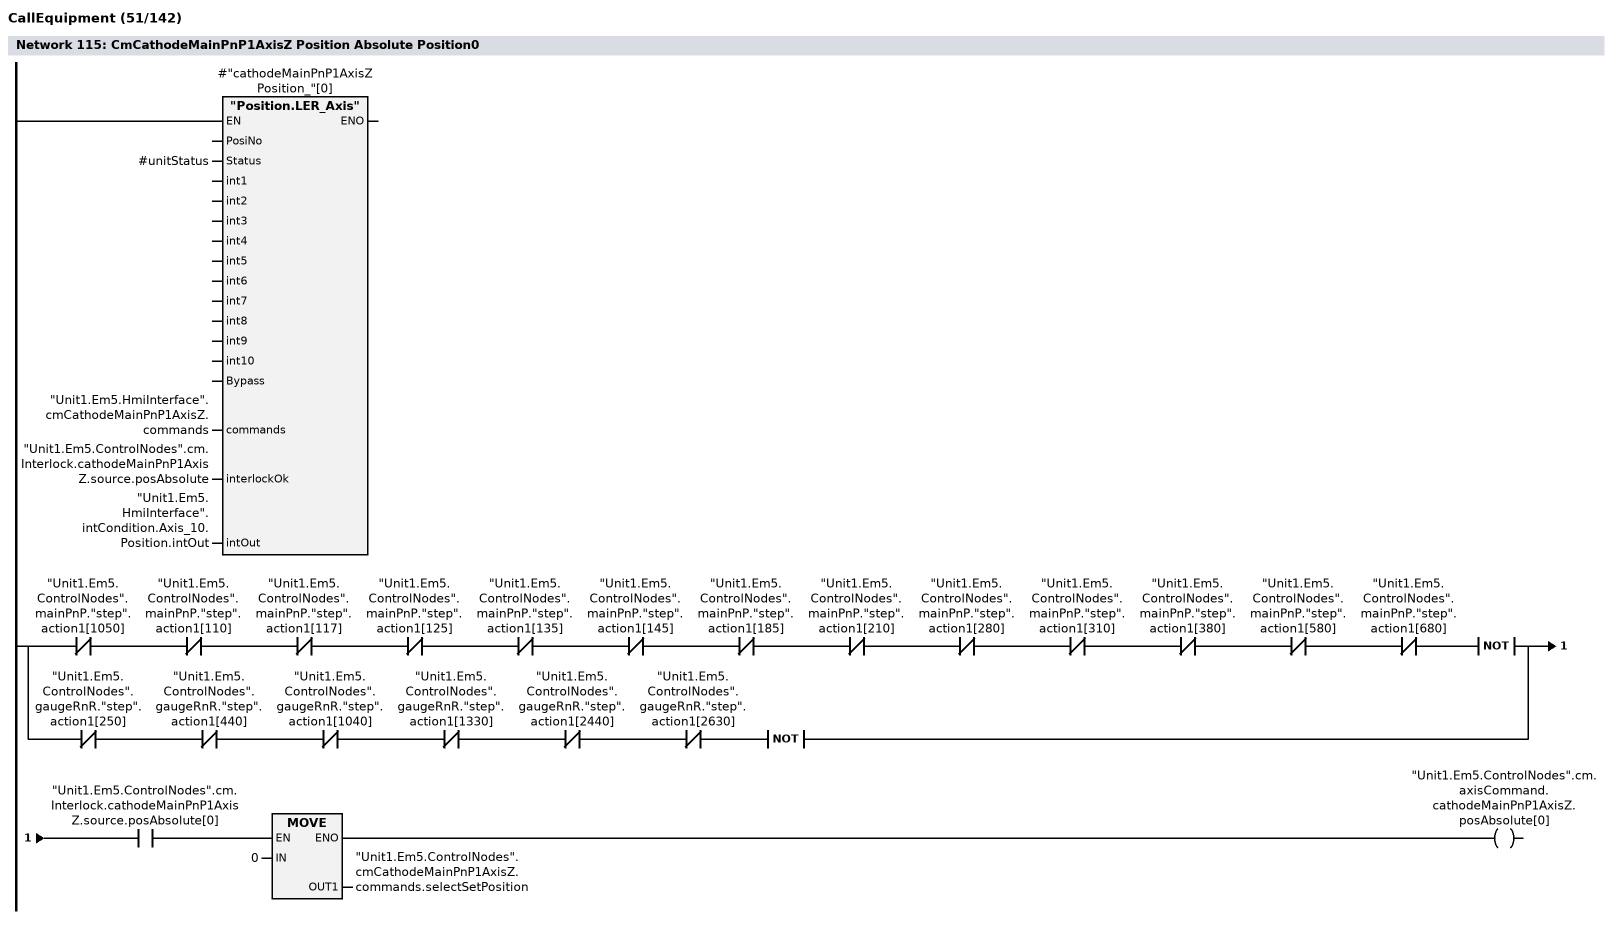
   RUNG wire#powerrail
      #"cathodeMainPnP1AxisZ Position_"[0](PosiNo :=, Status := #unitStatus, int1 :=, int2 :=, int3 :=, int4 :=, int5 :=, int6 :=, int7 :=, int8 :=, int9 :=, int10 :=, Bypass :=, commands := "Unit1.Em5.HmiInterface".cmCathodeMainPnP1AxisZ.commands, interlockOk := "Unit1.Em5.ControlNodes".cm.Interlock.cathodeMainPnP1AxisZ.source.posAbsolute, intOut := "Unit1.Em5.HmiInterface".intCondition.Axis_10.Position.intOut)
   END_RUNG
   RUNG wire#powerrail
      I_Contact( "Unit1.Em5.ControlNodes".mainPnP."step".action1[1050] )
      I_Contact( "Unit1.Em5.ControlNodes".mainPnP."step".action1[110] )
      I_Contact( "Unit1.Em5.ControlNodes".mainPnP."step".action1[117] )
      I_Contact( "Unit1.Em5.ControlNodes".mainPnP."step".action1[125] )
      I_Contact( "Unit1.Em5.ControlNodes".mainPnP."step".action1[135] )
      I_Contact( "Unit1.Em5.ControlNodes".mainPnP."step".action1[145] )
      I_Contact( "Unit1.Em5.ControlNodes".mainPnP."step".action1[185] )
      I_Contact( "Unit1.Em5.ControlNodes".mainPnP."step".action1[210] )
      I_Contact( "Unit1.Em5.ControlNodes".mainPnP."step".action1[280] )
      I_Contact( "Unit1.Em5.ControlNodes".mainPnP."step".action1[310] )
      I_Contact( "Unit1.Em5.ControlNodes".mainPnP."step".action1[380] )
      I_Contact( "Unit1.Em5.ControlNodes".mainPnP."step".action1[580] )
      I_Contact( "Unit1.Em5.ControlNodes".mainPnP."step".action1[680] )
      Not()
      wire#w1
      Contact( "Unit1.Em5.ControlNodes".cm.Interlock.cathodeMainPnP1AxisZ.source.posAbsolute[0] )
      Move(in := 0, out1 => "Unit1.Em5.ControlNodes".cmCathodeMainPnP1AxisZ.commands.selectSetPosition)
      Coil( "Unit1.Em5.ControlNodes".cm.axisCommand.cathodeMainPnP1AxisZ.posAbsolute[0] )
   END_RUNG
   RUNG wire#powerrail
      I_Contact( "Unit1.Em5.ControlNodes".gaugeRnR."step".action1[250] )
      I_Contact( "Unit1.Em5.ControlNodes".gaugeRnR."step".action1[440] )
      I_Contact( "Unit1.Em5.ControlNodes".gaugeRnR."step".action1[1040] )
      I_Contact( "Unit1.Em5.ControlNodes".gaugeRnR."step".action1[1330] )
      I_Contact( "Unit1.Em5.ControlNodes".gaugeRnR."step".action1[2440] )
      I_Contact( "Unit1.Em5.ControlNodes".gaugeRnR."step".action1[2630] )
      Not()
   END_RUNG wire#w1
   // the same network as SCL:
   #"cathodeMainPnP1AxisZ Position_"[0](Status := #unitStatus,   // "Position.LER_Axis"
                           commands := "Unit1.Em5.HmiInterface".cmCathodeMainPnP1AxisZ.commands,
                           interlockOk := "Unit1.Em5.ControlNodes".cm.Interlock.cathodeMainPnP1AxisZ.source.posAbsolute,
                           intOut := "Unit1.Em5.HmiInterface".intCondition.Axis_10.Position.intOut);
   #_w1 := (NOT (NOT "Unit1.Em5.ControlNodes".mainPnP."step".action1[1050] AND NOT "Unit1.Em5.ControlNodes".mainPnP."step".action1[110] AND NOT "Unit1.Em5.ControlNodes".mainPnP."step".action1[117] AND NOT "Unit1.Em5.ControlNodes".mainPnP."step".action1[125] AND NOT "Unit1.Em5.ControlNodes".mainPnP."step".action1[135] AND NOT "Unit1.Em5.ControlNodes".mainPnP."step".action1[145] AND NOT "Unit1.Em5.ControlNodes".mainPnP."step".action1[185] AND NOT "Unit1.Em5.ControlNodes".mainPnP."step".action1[210] AND NOT "Unit1.Em5.ControlNodes".mainPnP."step".action1[280] AND NOT "Unit1.Em5.ControlNodes".mainPnP."step".action1[310] AND NOT "Unit1.Em5.ControlNodes".mainPnP."step".action1[380] AND NOT "Unit1.Em5.ControlNodes".mainPnP."step".action1[580] AND NOT "Unit1.Em5.ControlNodes".mainPnP."step".action1[680]) OR NOT (NOT "Unit1.Em5.ControlNodes".gaugeRnR."step".action1[250] AND NOT "Unit1.Em5.ControlNodes".gaugeRnR."step".action1[440] AND NOT "Unit1.Em5.ControlNodes".gaugeRnR."step".action1[1040] AND NOT "Unit1.Em5.ControlNodes".gaugeRnR."step".action1[1330] AND NOT "Unit1.Em5.ControlNodes".gaugeRnR."step".action1[2440] AND NOT "Unit1.Em5.ControlNodes".gaugeRnR."step".action1[2630])) AND "Unit1.Em5.ControlNodes".cm.Interlock.cathodeMainPnP1AxisZ.source.posAbsolute[0];
   IF #_w1 THEN "Unit1.Em5.ControlNodes".cmCathodeMainPnP1AxisZ.commands.selectSetPosition := 0; END_IF;
   "Unit1.Em5.ControlNodes".cm.axisCommand.cathodeMainPnP1AxisZ.posAbsolute[0] := #_w1;
END_REGION

REGION Network 116: CmCathodeMainPnP1AxisZ Position Absolute Position1
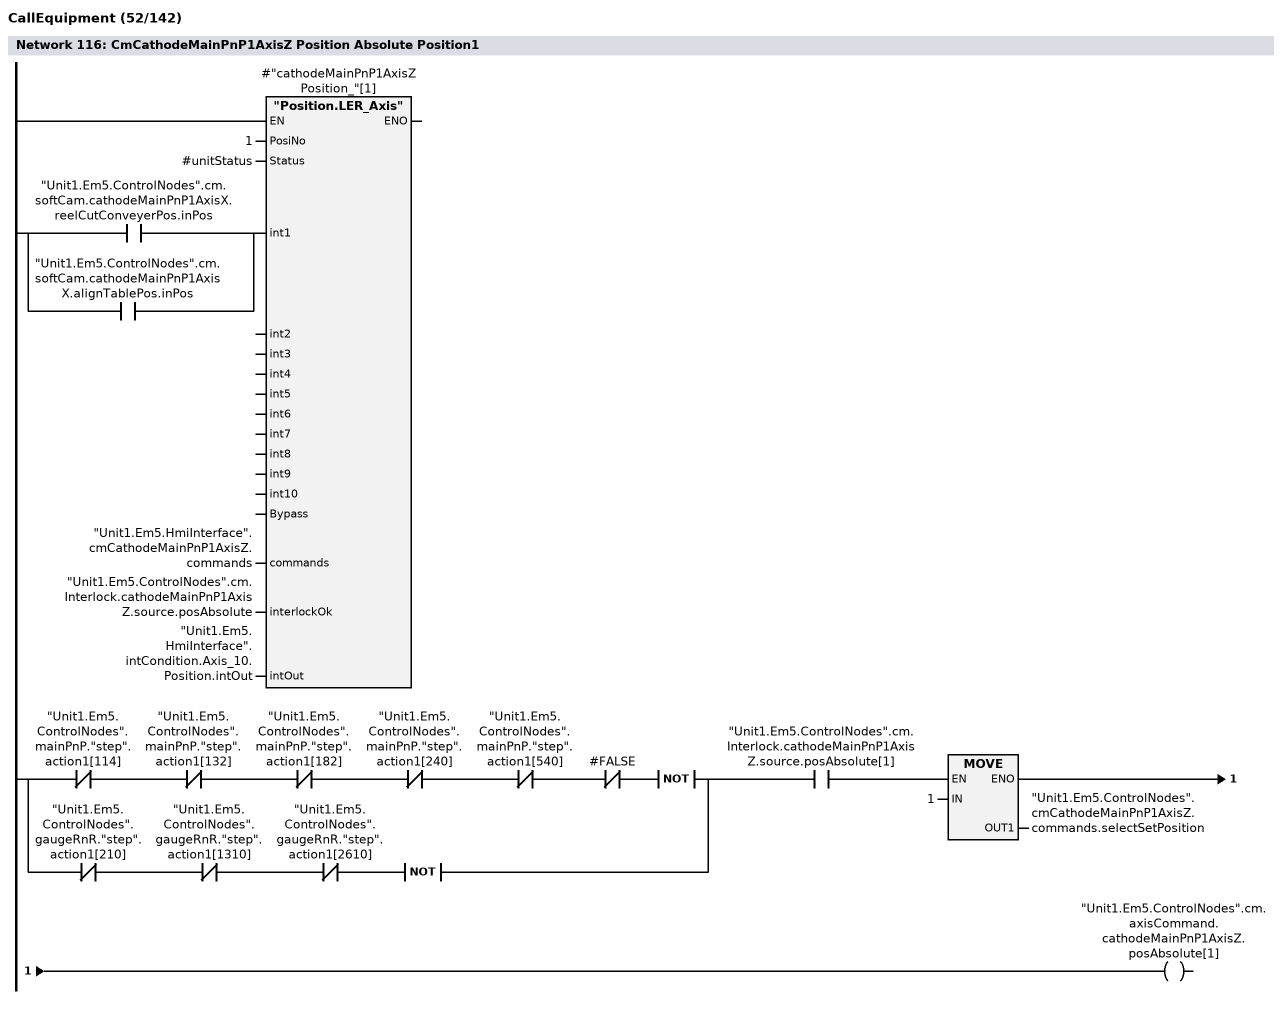
   RUNG wire#powerrail
      #"cathodeMainPnP1AxisZ Position_"[1](int1 := wire#w1, PosiNo := 1, Status := #unitStatus, int2 :=, int3 :=, int4 :=, int5 :=, int6 :=, int7 :=, int8 :=, int9 :=, int10 :=, Bypass :=, commands := "Unit1.Em5.HmiInterface".cmCathodeMainPnP1AxisZ.commands, interlockOk := "Unit1.Em5.ControlNodes".cm.Interlock.cathodeMainPnP1AxisZ.source.posAbsolute, intOut := "Unit1.Em5.HmiInterface".intCondition.Axis_10.Position.intOut)
   END_RUNG
   RUNG wire#powerrail
      Contact( "Unit1.Em5.ControlNodes".cm.softCam.cathodeMainPnP1AxisX.reelCutConveyerPos.inPos )
   END_RUNG wire#w1
   RUNG wire#powerrail
      Contact( "Unit1.Em5.ControlNodes".cm.softCam.cathodeMainPnP1AxisX.alignTablePos.inPos )
   END_RUNG wire#w1
   RUNG wire#powerrail
      I_Contact( "Unit1.Em5.ControlNodes".mainPnP."step".action1[114] )
      I_Contact( "Unit1.Em5.ControlNodes".mainPnP."step".action1[132] )
      I_Contact( "Unit1.Em5.ControlNodes".mainPnP."step".action1[182] )
      I_Contact( "Unit1.Em5.ControlNodes".mainPnP."step".action1[240] )
      I_Contact( "Unit1.Em5.ControlNodes".mainPnP."step".action1[540] )
      I_Contact( #FALSE )
      Not()
      wire#w2
      Contact( "Unit1.Em5.ControlNodes".cm.Interlock.cathodeMainPnP1AxisZ.source.posAbsolute[1] )
      Move(in := 1, out1 => "Unit1.Em5.ControlNodes".cmCathodeMainPnP1AxisZ.commands.selectSetPosition)
      Coil( "Unit1.Em5.ControlNodes".cm.axisCommand.cathodeMainPnP1AxisZ.posAbsolute[1] )
   END_RUNG
   RUNG wire#powerrail
      I_Contact( "Unit1.Em5.ControlNodes".gaugeRnR."step".action1[210] )
      I_Contact( "Unit1.Em5.ControlNodes".gaugeRnR."step".action1[1310] )
      I_Contact( "Unit1.Em5.ControlNodes".gaugeRnR."step".action1[2610] )
      Not()
   END_RUNG wire#w2
   // the same network as SCL:
   #"cathodeMainPnP1AxisZ Position_"[1](PosiNo := 1,   // "Position.LER_Axis"
                           Status := #unitStatus,
                           int1 := "Unit1.Em5.ControlNodes".cm.softCam.cathodeMainPnP1AxisX.reelCutConveyerPos.inPos OR "Unit1.Em5.ControlNodes".cm.softCam.cathodeMainPnP1AxisX.alignTablePos.inPos,
                           commands := "Unit1.Em5.HmiInterface".cmCathodeMainPnP1AxisZ.commands,
                           interlockOk := "Unit1.Em5.ControlNodes".cm.Interlock.cathodeMainPnP1AxisZ.source.posAbsolute,
                           intOut := "Unit1.Em5.HmiInterface".intCondition.Axis_10.Position.intOut);
   #_w1 := (NOT (NOT "Unit1.Em5.ControlNodes".mainPnP."step".action1[114] AND NOT "Unit1.Em5.ControlNodes".mainPnP."step".action1[132] AND NOT "Unit1.Em5.ControlNodes".mainPnP."step".action1[182] AND NOT "Unit1.Em5.ControlNodes".mainPnP."step".action1[240] AND NOT "Unit1.Em5.ControlNodes".mainPnP."step".action1[540] AND NOT #FALSE) OR NOT (NOT "Unit1.Em5.ControlNodes".gaugeRnR."step".action1[210] AND NOT "Unit1.Em5.ControlNodes".gaugeRnR."step".action1[1310] AND NOT "Unit1.Em5.ControlNodes".gaugeRnR."step".action1[2610])) AND "Unit1.Em5.ControlNodes".cm.Interlock.cathodeMainPnP1AxisZ.source.posAbsolute[1];
   IF #_w1 THEN "Unit1.Em5.ControlNodes".cmCathodeMainPnP1AxisZ.commands.selectSetPosition := 1; END_IF;
   "Unit1.Em5.ControlNodes".cm.axisCommand.cathodeMainPnP1AxisZ.posAbsolute[1] := #_w1;
END_REGION

REGION Network 117: CmCathodeMainPnP1AxisZ Position Absolute Position2
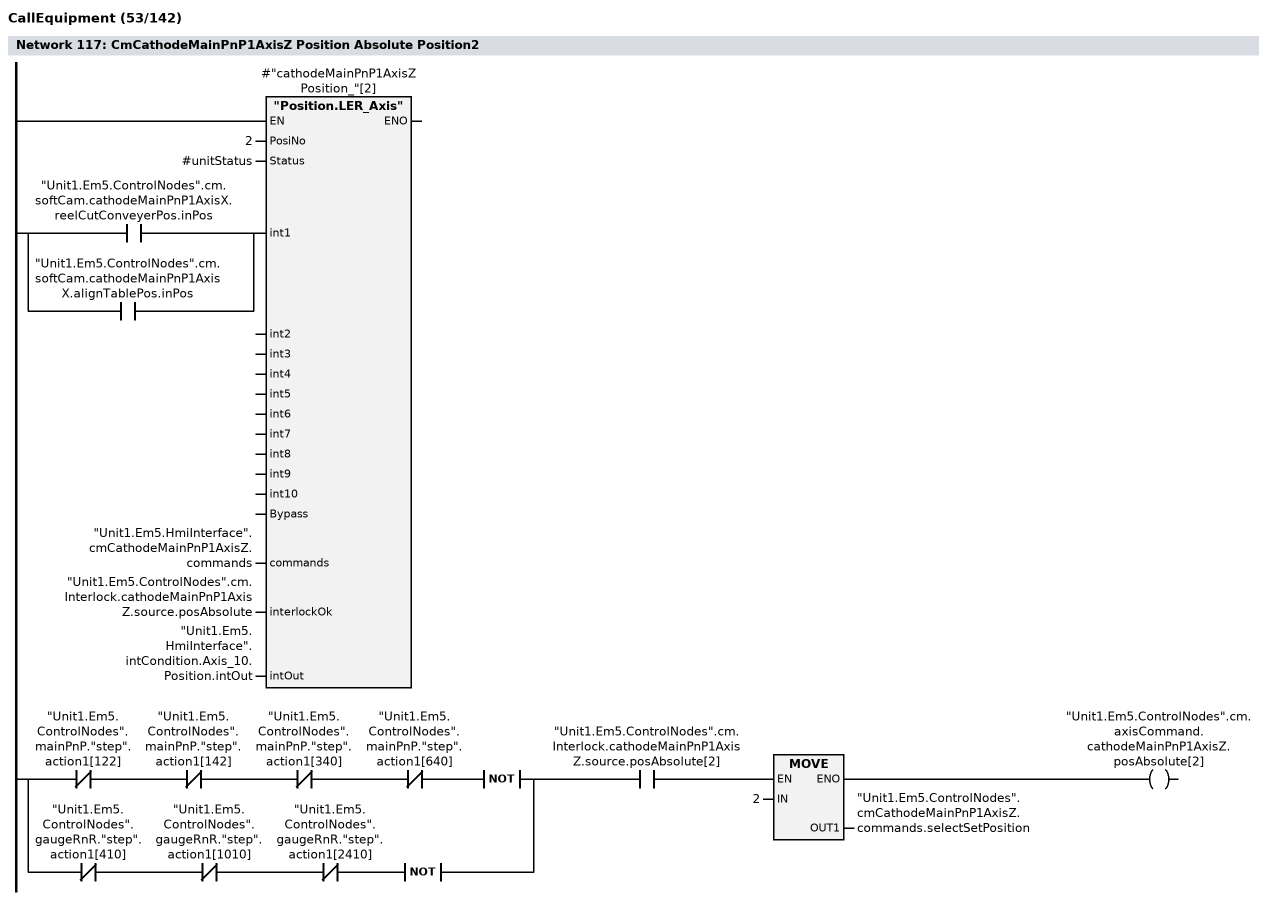
   RUNG wire#powerrail
      #"cathodeMainPnP1AxisZ Position_"[2](int1 := wire#w1, PosiNo := 2, Status := #unitStatus, int2 :=, int3 :=, int4 :=, int5 :=, int6 :=, int7 :=, int8 :=, int9 :=, int10 :=, Bypass :=, commands := "Unit1.Em5.HmiInterface".cmCathodeMainPnP1AxisZ.commands, interlockOk := "Unit1.Em5.ControlNodes".cm.Interlock.cathodeMainPnP1AxisZ.source.posAbsolute, intOut := "Unit1.Em5.HmiInterface".intCondition.Axis_10.Position.intOut)
   END_RUNG
   RUNG wire#powerrail
      Contact( "Unit1.Em5.ControlNodes".cm.softCam.cathodeMainPnP1AxisX.reelCutConveyerPos.inPos )
   END_RUNG wire#w1
   RUNG wire#powerrail
      Contact( "Unit1.Em5.ControlNodes".cm.softCam.cathodeMainPnP1AxisX.alignTablePos.inPos )
   END_RUNG wire#w1
   RUNG wire#powerrail
      I_Contact( "Unit1.Em5.ControlNodes".mainPnP."step".action1[122] )
      I_Contact( "Unit1.Em5.ControlNodes".mainPnP."step".action1[142] )
      I_Contact( "Unit1.Em5.ControlNodes".mainPnP."step".action1[340] )
      I_Contact( "Unit1.Em5.ControlNodes".mainPnP."step".action1[640] )
      Not()
      wire#w2
      Contact( "Unit1.Em5.ControlNodes".cm.Interlock.cathodeMainPnP1AxisZ.source.posAbsolute[2] )
      Move(in := 2, out1 => "Unit1.Em5.ControlNodes".cmCathodeMainPnP1AxisZ.commands.selectSetPosition)
      Coil( "Unit1.Em5.ControlNodes".cm.axisCommand.cathodeMainPnP1AxisZ.posAbsolute[2] )
   END_RUNG
   RUNG wire#powerrail
      I_Contact( "Unit1.Em5.ControlNodes".gaugeRnR."step".action1[410] )
      I_Contact( "Unit1.Em5.ControlNodes".gaugeRnR."step".action1[1010] )
      I_Contact( "Unit1.Em5.ControlNodes".gaugeRnR."step".action1[2410] )
      Not()
   END_RUNG wire#w2
   // the same network as SCL:
   #"cathodeMainPnP1AxisZ Position_"[2](PosiNo := 2,   // "Position.LER_Axis"
                           Status := #unitStatus,
                           int1 := "Unit1.Em5.ControlNodes".cm.softCam.cathodeMainPnP1AxisX.reelCutConveyerPos.inPos OR "Unit1.Em5.ControlNodes".cm.softCam.cathodeMainPnP1AxisX.alignTablePos.inPos,
                           commands := "Unit1.Em5.HmiInterface".cmCathodeMainPnP1AxisZ.commands,
                           interlockOk := "Unit1.Em5.ControlNodes".cm.Interlock.cathodeMainPnP1AxisZ.source.posAbsolute,
                           intOut := "Unit1.Em5.HmiInterface".intCondition.Axis_10.Position.intOut);
   #_w1 := (NOT (NOT "Unit1.Em5.ControlNodes".mainPnP."step".action1[122] AND NOT "Unit1.Em5.ControlNodes".mainPnP."step".action1[142] AND NOT "Unit1.Em5.ControlNodes".mainPnP."step".action1[340] AND NOT "Unit1.Em5.ControlNodes".mainPnP."step".action1[640]) OR NOT (NOT "Unit1.Em5.ControlNodes".gaugeRnR."step".action1[410] AND NOT "Unit1.Em5.ControlNodes".gaugeRnR."step".action1[1010] AND NOT "Unit1.Em5.ControlNodes".gaugeRnR."step".action1[2410])) AND "Unit1.Em5.ControlNodes".cm.Interlock.cathodeMainPnP1AxisZ.source.posAbsolute[2];
   IF #_w1 THEN "Unit1.Em5.ControlNodes".cmCathodeMainPnP1AxisZ.commands.selectSetPosition := 2; END_IF;
   "Unit1.Em5.ControlNodes".cm.axisCommand.cathodeMainPnP1AxisZ.posAbsolute[2] := #_w1;
END_REGION

REGION Network 118: CmCathodeMainPnP1AxisZ Position Absolute Position3
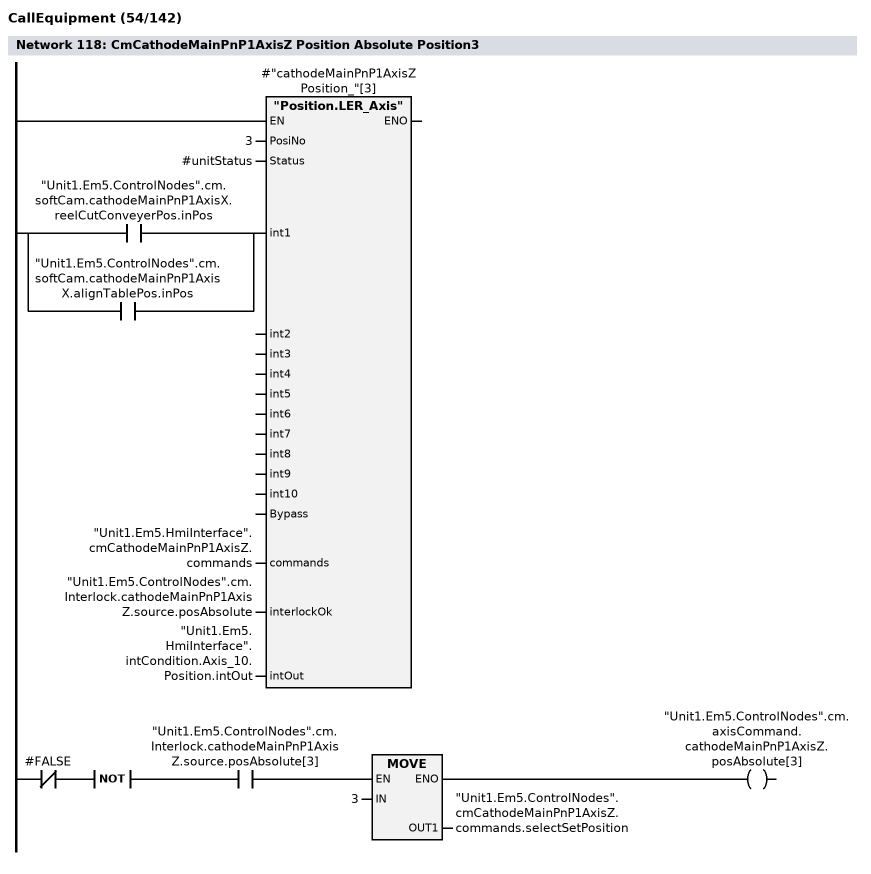
   RUNG wire#powerrail
      #"cathodeMainPnP1AxisZ Position_"[3](int1 := wire#w1, PosiNo := 3, Status := #unitStatus, int2 :=, int3 :=, int4 :=, int5 :=, int6 :=, int7 :=, int8 :=, int9 :=, int10 :=, Bypass :=, commands := "Unit1.Em5.HmiInterface".cmCathodeMainPnP1AxisZ.commands, interlockOk := "Unit1.Em5.ControlNodes".cm.Interlock.cathodeMainPnP1AxisZ.source.posAbsolute, intOut := "Unit1.Em5.HmiInterface".intCondition.Axis_10.Position.intOut)
   END_RUNG
   RUNG wire#powerrail
      Contact( "Unit1.Em5.ControlNodes".cm.softCam.cathodeMainPnP1AxisX.reelCutConveyerPos.inPos )
   END_RUNG wire#w1
   RUNG wire#powerrail
      Contact( "Unit1.Em5.ControlNodes".cm.softCam.cathodeMainPnP1AxisX.alignTablePos.inPos )
   END_RUNG wire#w1
   RUNG wire#powerrail
      I_Contact( #FALSE )
      Not()
      Contact( "Unit1.Em5.ControlNodes".cm.Interlock.cathodeMainPnP1AxisZ.source.posAbsolute[3] )
      Move(in := 3, out1 => "Unit1.Em5.ControlNodes".cmCathodeMainPnP1AxisZ.commands.selectSetPosition)
      Coil( "Unit1.Em5.ControlNodes".cm.axisCommand.cathodeMainPnP1AxisZ.posAbsolute[3] )
   END_RUNG
   // the same network as SCL:
   #"cathodeMainPnP1AxisZ Position_"[3](PosiNo := 3,   // "Position.LER_Axis"
                           Status := #unitStatus,
                           int1 := "Unit1.Em5.ControlNodes".cm.softCam.cathodeMainPnP1AxisX.reelCutConveyerPos.inPos OR "Unit1.Em5.ControlNodes".cm.softCam.cathodeMainPnP1AxisX.alignTablePos.inPos,
                           commands := "Unit1.Em5.HmiInterface".cmCathodeMainPnP1AxisZ.commands,
                           interlockOk := "Unit1.Em5.ControlNodes".cm.Interlock.cathodeMainPnP1AxisZ.source.posAbsolute,
                           intOut := "Unit1.Em5.HmiInterface".intCondition.Axis_10.Position.intOut);
   #_w1 := NOT (NOT #FALSE) AND "Unit1.Em5.ControlNodes".cm.Interlock.cathodeMainPnP1AxisZ.source.posAbsolute[3];
   IF #_w1 THEN "Unit1.Em5.ControlNodes".cmCathodeMainPnP1AxisZ.commands.selectSetPosition := 3; END_IF;
   "Unit1.Em5.ControlNodes".cm.axisCommand.cathodeMainPnP1AxisZ.posAbsolute[3] := #_w1;
END_REGION

REGION Network 119: CmCathodeMainPnP1AxisZ Position Absolute Position4
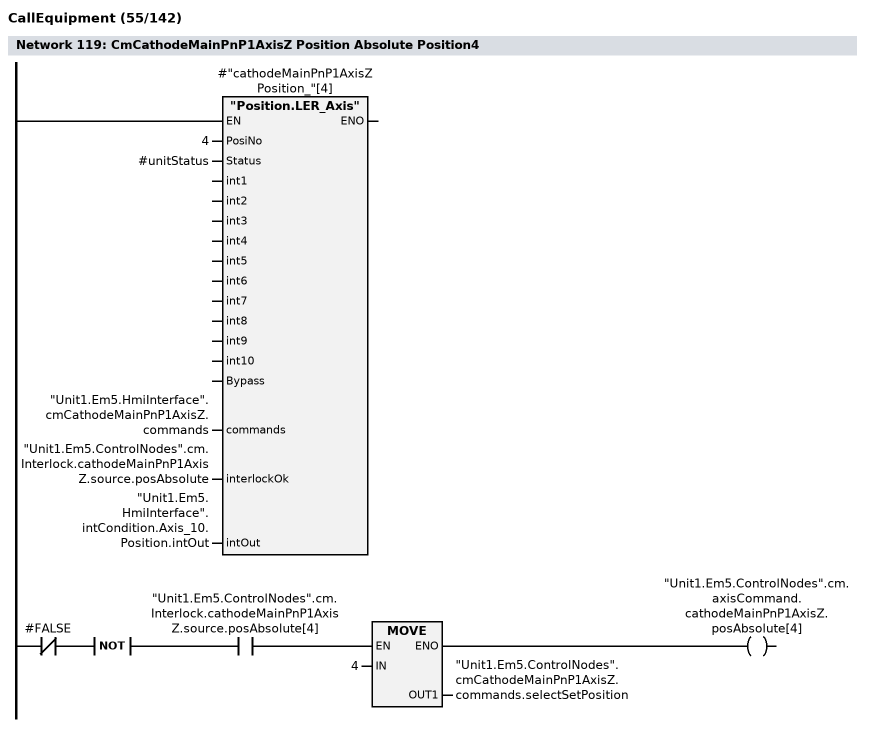
   RUNG wire#powerrail
      #"cathodeMainPnP1AxisZ Position_"[4](PosiNo := 4, Status := #unitStatus, int1 :=, int2 :=, int3 :=, int4 :=, int5 :=, int6 :=, int7 :=, int8 :=, int9 :=, int10 :=, Bypass :=, commands := "Unit1.Em5.HmiInterface".cmCathodeMainPnP1AxisZ.commands, interlockOk := "Unit1.Em5.ControlNodes".cm.Interlock.cathodeMainPnP1AxisZ.source.posAbsolute, intOut := "Unit1.Em5.HmiInterface".intCondition.Axis_10.Position.intOut)
   END_RUNG
   RUNG wire#powerrail
      I_Contact( #FALSE )
      Not()
      Contact( "Unit1.Em5.ControlNodes".cm.Interlock.cathodeMainPnP1AxisZ.source.posAbsolute[4] )
      Move(in := 4, out1 => "Unit1.Em5.ControlNodes".cmCathodeMainPnP1AxisZ.commands.selectSetPosition)
      Coil( "Unit1.Em5.ControlNodes".cm.axisCommand.cathodeMainPnP1AxisZ.posAbsolute[4] )
   END_RUNG
   // the same network as SCL:
   #"cathodeMainPnP1AxisZ Position_"[4](PosiNo := 4,   // "Position.LER_Axis"
                           Status := #unitStatus,
                           commands := "Unit1.Em5.HmiInterface".cmCathodeMainPnP1AxisZ.commands,
                           interlockOk := "Unit1.Em5.ControlNodes".cm.Interlock.cathodeMainPnP1AxisZ.source.posAbsolute,
                           intOut := "Unit1.Em5.HmiInterface".intCondition.Axis_10.Position.intOut);
   #_w1 := NOT (NOT #FALSE) AND "Unit1.Em5.ControlNodes".cm.Interlock.cathodeMainPnP1AxisZ.source.posAbsolute[4];
   IF #_w1 THEN "Unit1.Em5.ControlNodes".cmCathodeMainPnP1AxisZ.commands.selectSetPosition := 4; END_IF;
   "Unit1.Em5.ControlNodes".cm.axisCommand.cathodeMainPnP1AxisZ.posAbsolute[4] := #_w1;
END_REGION

REGION Network 120: CmCathodeMainPnP1AxisZ Position Absolute Position5
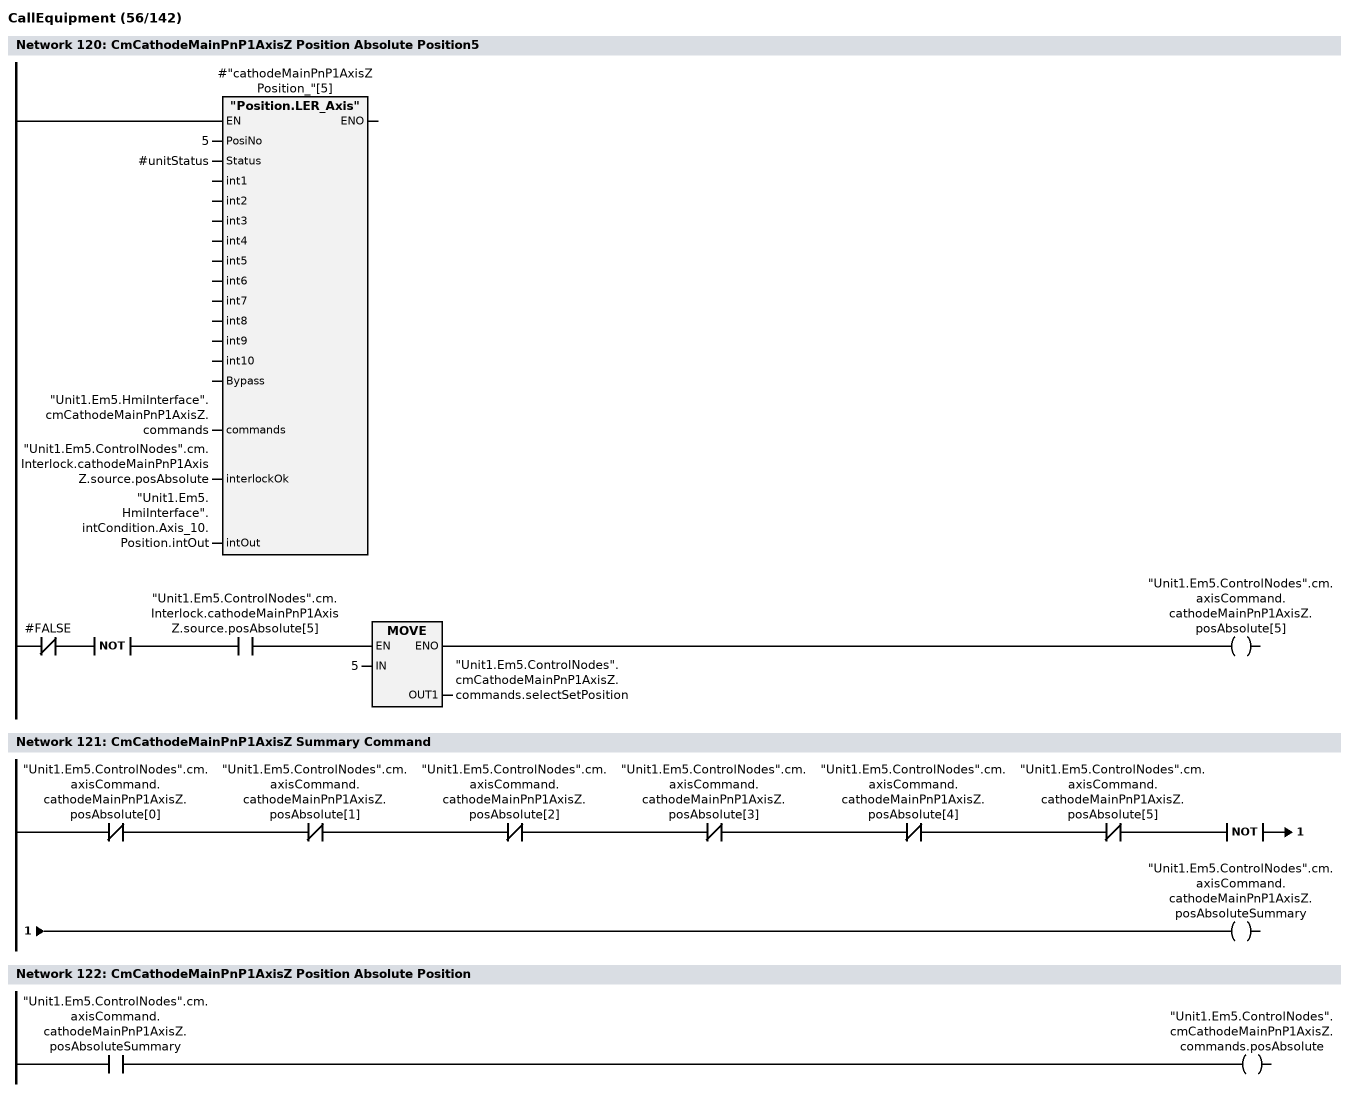
   RUNG wire#powerrail
      #"cathodeMainPnP1AxisZ Position_"[5](PosiNo := 5, Status := #unitStatus, int1 :=, int2 :=, int3 :=, int4 :=, int5 :=, int6 :=, int7 :=, int8 :=, int9 :=, int10 :=, Bypass :=, commands := "Unit1.Em5.HmiInterface".cmCathodeMainPnP1AxisZ.commands, interlockOk := "Unit1.Em5.ControlNodes".cm.Interlock.cathodeMainPnP1AxisZ.source.posAbsolute, intOut := "Unit1.Em5.HmiInterface".intCondition.Axis_10.Position.intOut)
   END_RUNG
   RUNG wire#powerrail
      I_Contact( #FALSE )
      Not()
      Contact( "Unit1.Em5.ControlNodes".cm.Interlock.cathodeMainPnP1AxisZ.source.posAbsolute[5] )
      Move(in := 5, out1 => "Unit1.Em5.ControlNodes".cmCathodeMainPnP1AxisZ.commands.selectSetPosition)
      Coil( "Unit1.Em5.ControlNodes".cm.axisCommand.cathodeMainPnP1AxisZ.posAbsolute[5] )
   END_RUNG
   // the same network as SCL:
   #"cathodeMainPnP1AxisZ Position_"[5](PosiNo := 5,   // "Position.LER_Axis"
                           Status := #unitStatus,
                           commands := "Unit1.Em5.HmiInterface".cmCathodeMainPnP1AxisZ.commands,
                           interlockOk := "Unit1.Em5.ControlNodes".cm.Interlock.cathodeMainPnP1AxisZ.source.posAbsolute,
                           intOut := "Unit1.Em5.HmiInterface".intCondition.Axis_10.Position.intOut);
   #_w1 := NOT (NOT #FALSE) AND "Unit1.Em5.ControlNodes".cm.Interlock.cathodeMainPnP1AxisZ.source.posAbsolute[5];
   IF #_w1 THEN "Unit1.Em5.ControlNodes".cmCathodeMainPnP1AxisZ.commands.selectSetPosition := 5; END_IF;
   "Unit1.Em5.ControlNodes".cm.axisCommand.cathodeMainPnP1AxisZ.posAbsolute[5] := #_w1;
END_REGION

REGION Network 121: CmCathodeMainPnP1AxisZ Summary Command
   RUNG wire#powerrail
      I_Contact( "Unit1.Em5.ControlNodes".cm.axisCommand.cathodeMainPnP1AxisZ.posAbsolute[0] )
      I_Contact( "Unit1.Em5.ControlNodes".cm.axisCommand.cathodeMainPnP1AxisZ.posAbsolute[1] )
      I_Contact( "Unit1.Em5.ControlNodes".cm.axisCommand.cathodeMainPnP1AxisZ.posAbsolute[2] )
      I_Contact( "Unit1.Em5.ControlNodes".cm.axisCommand.cathodeMainPnP1AxisZ.posAbsolute[3] )
      I_Contact( "Unit1.Em5.ControlNodes".cm.axisCommand.cathodeMainPnP1AxisZ.posAbsolute[4] )
      I_Contact( "Unit1.Em5.ControlNodes".cm.axisCommand.cathodeMainPnP1AxisZ.posAbsolute[5] )
      Not()
      Coil( "Unit1.Em5.ControlNodes".cm.axisCommand.cathodeMainPnP1AxisZ.posAbsoluteSummary )
   END_RUNG
   // the same network as SCL:
   "Unit1.Em5.ControlNodes".cm.axisCommand.cathodeMainPnP1AxisZ.posAbsoluteSummary := NOT (NOT "Unit1.Em5.ControlNodes".cm.axisCommand.cathodeMainPnP1AxisZ.posAbsolute[0] AND NOT "Unit1.Em5.ControlNodes".cm.axisCommand.cathodeMainPnP1AxisZ.posAbsolute[1] AND NOT "Unit1.Em5.ControlNodes".cm.axisCommand.cathodeMainPnP1AxisZ.posAbsolute[2] AND NOT "Unit1.Em5.ControlNodes".cm.axisCommand.cathodeMainPnP1AxisZ.posAbsolute[3] AND NOT "Unit1.Em5.ControlNodes".cm.axisCommand.cathodeMainPnP1AxisZ.posAbsolute[4] AND NOT "Unit1.Em5.ControlNodes".cm.axisCommand.cathodeMainPnP1AxisZ.posAbsolute[5]);
END_REGION

REGION Network 122: CmCathodeMainPnP1AxisZ Position Absolute Position
   RUNG wire#powerrail
      Contact( "Unit1.Em5.ControlNodes".cm.axisCommand.cathodeMainPnP1AxisZ.posAbsoluteSummary )
      Coil( "Unit1.Em5.ControlNodes".cmCathodeMainPnP1AxisZ.commands.posAbsolute )
   END_RUNG
   // the same network as SCL:
   "Unit1.Em5.ControlNodes".cmCathodeMainPnP1AxisZ.commands.posAbsolute := "Unit1.Em5.ControlNodes".cm.axisCommand.cathodeMainPnP1AxisZ.posAbsoluteSummary;
END_REGION

REGION Network 123: CmCathodeMainPnP1AxisZ Interlock Summary
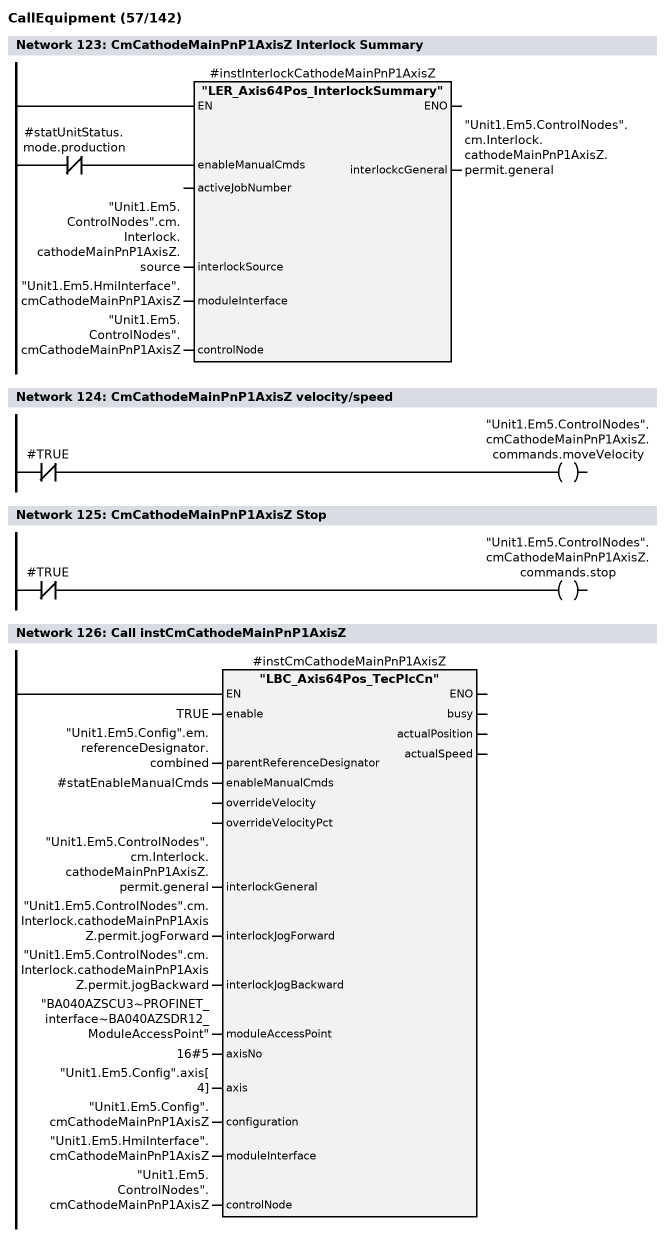
   RUNG wire#powerrail
      #instInterlockCathodeMainPnP1AxisZ(enableManualCmds := wire#w1, activeJobNumber :=, interlockSource := "Unit1.Em5.ControlNodes".cm.Interlock.cathodeMainPnP1AxisZ.source, moduleInterface := "Unit1.Em5.HmiInterface".cmCathodeMainPnP1AxisZ, controlNode := "Unit1.Em5.ControlNodes".cmCathodeMainPnP1AxisZ, interlockcGeneral => "Unit1.Em5.ControlNodes".cm.Interlock.cathodeMainPnP1AxisZ.permit.general)
   END_RUNG
   RUNG wire#powerrail
      I_Contact( #statUnitStatus.mode.production )
   END_RUNG wire#w1
   // the same network as SCL:
   #instInterlockCathodeMainPnP1AxisZ(enableManualCmds := NOT #statUnitStatus.mode.production,   // "LER_Axis64Pos_InterlockSummary"
                           interlockSource := "Unit1.Em5.ControlNodes".cm.Interlock.cathodeMainPnP1AxisZ.source,
                           moduleInterface := "Unit1.Em5.HmiInterface".cmCathodeMainPnP1AxisZ,
                           controlNode := "Unit1.Em5.ControlNodes".cmCathodeMainPnP1AxisZ,
                           interlockcGeneral => "Unit1.Em5.ControlNodes".cm.Interlock.cathodeMainPnP1AxisZ.permit.general);
END_REGION

REGION Network 124: CmCathodeMainPnP1AxisZ velocity/speed
   RUNG wire#powerrail
      I_Contact( #TRUE )
      Coil( "Unit1.Em5.ControlNodes".cmCathodeMainPnP1AxisZ.commands.moveVelocity )
   END_RUNG
   // the same network as SCL:
   "Unit1.Em5.ControlNodes".cmCathodeMainPnP1AxisZ.commands.moveVelocity := NOT #TRUE;
END_REGION

REGION Network 125: CmCathodeMainPnP1AxisZ Stop
   RUNG wire#powerrail
      I_Contact( #TRUE )
      Coil( "Unit1.Em5.ControlNodes".cmCathodeMainPnP1AxisZ.commands.stop )
   END_RUNG
   // the same network as SCL:
   "Unit1.Em5.ControlNodes".cmCathodeMainPnP1AxisZ.commands.stop := NOT #TRUE;
END_REGION

REGION Network 126: Call instCmCathodeMainPnP1AxisZ
   RUNG wire#powerrail
      #instCmCathodeMainPnP1AxisZ(enable := TRUE, parentReferenceDesignator := "Unit1.Em5.Config".em.referenceDesignator.combined, enableManualCmds := #statEnableManualCmds, overrideVelocity :=, overrideVelocityPct :=, interlockGeneral := "Unit1.Em5.ControlNodes".cm.Interlock.cathodeMainPnP1AxisZ.permit.general, interlockJogForward := "Unit1.Em5.ControlNodes".cm.Interlock.cathodeMainPnP1AxisZ.permit.jogForward, interlockJogBackward := "Unit1.Em5.ControlNodes".cm.Interlock.cathodeMainPnP1AxisZ.permit.jogBackward, moduleAccessPoint := "BA040AZSCU3~PROFINET_interface~BA040AZSDR12_ModuleAccessPoint", axisNo := 16#5, axis := "Unit1.Em5.Config".axis[4], configuration := "Unit1.Em5.Config".cmCathodeMainPnP1AxisZ, moduleInterface := "Unit1.Em5.HmiInterface".cmCathodeMainPnP1AxisZ, controlNode := "Unit1.Em5.ControlNodes".cmCathodeMainPnP1AxisZ, busy =>, actualPosition =>, actualSpeed =>)
   END_RUNG
   // the same network as SCL:
   #instCmCathodeMainPnP1AxisZ(enable := TRUE,   // "LBC_Axis64Pos_TecPlcCn"
                           parentReferenceDesignator := "Unit1.Em5.Config".em.referenceDesignator.combined,
                           enableManualCmds := #statEnableManualCmds,
                           interlockGeneral := "Unit1.Em5.ControlNodes".cm.Interlock.cathodeMainPnP1AxisZ.permit.general,
                           interlockJogForward := "Unit1.Em5.ControlNodes".cm.Interlock.cathodeMainPnP1AxisZ.permit.jogForward,
                           interlockJogBackward := "Unit1.Em5.ControlNodes".cm.Interlock.cathodeMainPnP1AxisZ.permit.jogBackward,
                           moduleAccessPoint := "BA040AZSCU3~PROFINET_interface~BA040AZSDR12_ModuleAccessPoint",
                           axisNo := 16#5,
                           axis := "Unit1.Em5.Config".axis[4],
                           configuration := "Unit1.Em5.Config".cmCathodeMainPnP1AxisZ,
                           moduleInterface := "Unit1.Em5.HmiInterface".cmCathodeMainPnP1AxisZ,
                           controlNode := "Unit1.Em5.ControlNodes".cmCathodeMainPnP1AxisZ);
END_REGION

REGION Network 127: CmCathodeMainPnP1AxisY SoftCam
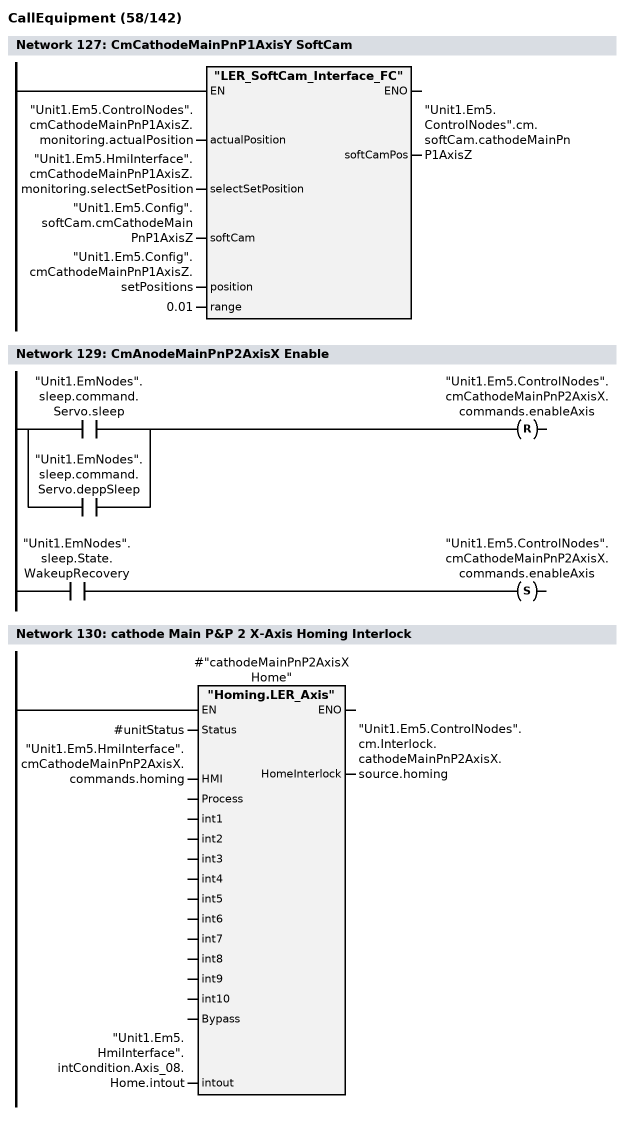
   RUNG wire#powerrail
      "LER_SoftCam_Interface_FC"(actualPosition := "Unit1.Em5.ControlNodes".cmCathodeMainPnP1AxisZ.monitoring.actualPosition, selectSetPosition := "Unit1.Em5.HmiInterface".cmCathodeMainPnP1AxisZ.monitoring.selectSetPosition, softCam := "Unit1.Em5.Config".softCam.cmCathodeMainPnP1AxisZ, position := "Unit1.Em5.Config".cmCathodeMainPnP1AxisZ.setPositions, range := 0.01, softCamPos => "Unit1.Em5.ControlNodes".cm.softCam.cathodeMainPnP1AxisZ)
   END_RUNG
   // the same network as SCL:
   "LER_SoftCam_Interface_FC"(actualPosition := "Unit1.Em5.ControlNodes".cmCathodeMainPnP1AxisZ.monitoring.actualPosition,
                           selectSetPosition := "Unit1.Em5.HmiInterface".cmCathodeMainPnP1AxisZ.monitoring.selectSetPosition,
                           softCam := "Unit1.Em5.Config".softCam.cmCathodeMainPnP1AxisZ,
                           position := "Unit1.Em5.Config".cmCathodeMainPnP1AxisZ.setPositions,
                           range := 0.01,
                           softCamPos => "Unit1.Em5.ControlNodes".cm.softCam.cathodeMainPnP1AxisZ);
END_REGION

REGION Network 129: CmAnodeMainPnP2AxisX Enable
   RUNG wire#powerrail
      Contact( "Unit1.EmNodes".sleep.command.Servo.sleep )
      wire#w1
      R_Coil( "Unit1.Em5.ControlNodes".cmCathodeMainPnP2AxisX.commands.enableAxis )
   END_RUNG
   RUNG wire#powerrail
      Contact( "Unit1.EmNodes".sleep.command.Servo.deppSleep )
   END_RUNG wire#w1
   RUNG wire#powerrail
      Contact( "Unit1.EmNodes".sleep.State.WakeupRecovery )
      S_Coil( "Unit1.Em5.ControlNodes".cmCathodeMainPnP2AxisX.commands.enableAxis )
   END_RUNG
   // the same network as SCL:
   IF "Unit1.EmNodes".sleep.command.Servo.sleep OR "Unit1.EmNodes".sleep.command.Servo.deppSleep THEN
       "Unit1.Em5.ControlNodes".cmCathodeMainPnP2AxisX.commands.enableAxis := FALSE;
   END_IF;
   IF "Unit1.EmNodes".sleep.State.WakeupRecovery THEN
       "Unit1.Em5.ControlNodes".cmCathodeMainPnP2AxisX.commands.enableAxis := TRUE;
   END_IF;
END_REGION

REGION Network 130: cathode Main P&P 2 X-Axis Homing Interlock
   RUNG wire#powerrail
      #"cathodeMainPnP2AxisX Home"(Status := #unitStatus, HMI := "Unit1.Em5.HmiInterface".cmCathodeMainPnP2AxisX.commands.homing, Process :=, int1 :=, int2 :=, int3 :=, int4 :=, int5 :=, int6 :=, int7 :=, int8 :=, int9 :=, int10 :=, Bypass :=, intout := "Unit1.Em5.HmiInterface".intCondition.Axis_08.Home.intout, HomeInterlock => "Unit1.Em5.ControlNodes".cm.Interlock.cathodeMainPnP2AxisX.source.homing)
   END_RUNG
   // the same network as SCL:
   #"cathodeMainPnP2AxisX Home"(Status := #unitStatus,   // "Homing.LER_Axis"
                           HMI := "Unit1.Em5.HmiInterface".cmCathodeMainPnP2AxisX.commands.homing,
                           intout := "Unit1.Em5.HmiInterface".intCondition.Axis_08.Home.intout,
                           HomeInterlock => "Unit1.Em5.ControlNodes".cm.Interlock.cathodeMainPnP2AxisX.source.homing);
END_REGION

REGION Network 131: CmCathodeMainPnP2AxisX Position Absolute Jog
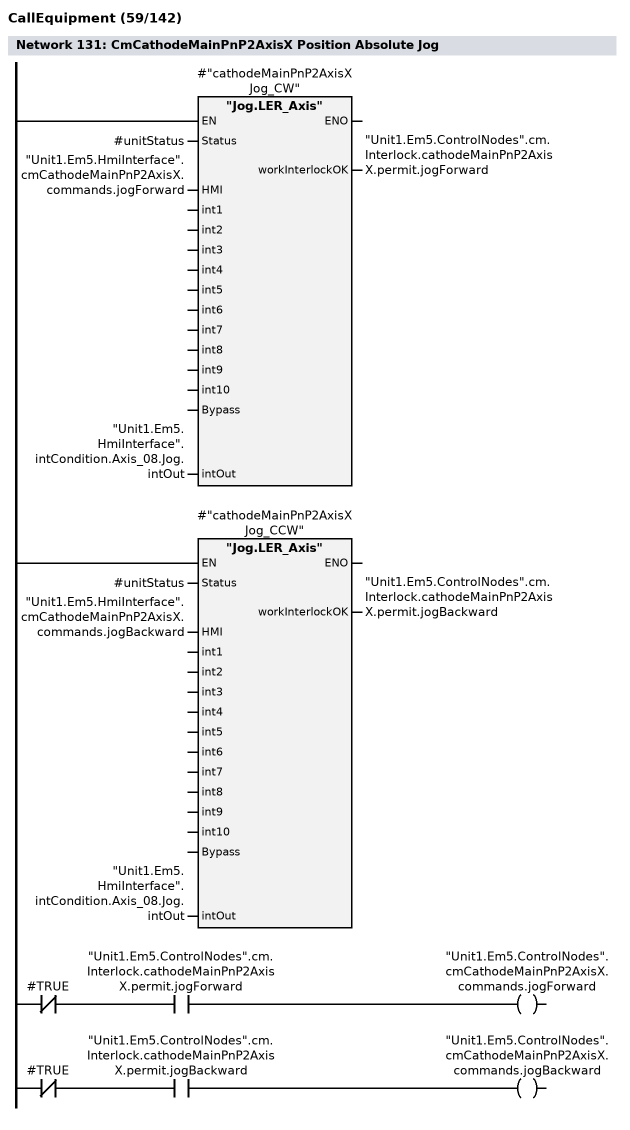
   RUNG wire#powerrail
      #"cathodeMainPnP2AxisX Jog_CW"(Status := #unitStatus, HMI := "Unit1.Em5.HmiInterface".cmCathodeMainPnP2AxisX.commands.jogForward, int1 :=, int2 :=, int3 :=, int4 :=, int5 :=, int6 :=, int7 :=, int8 :=, int9 :=, int10 :=, Bypass :=, intOut := "Unit1.Em5.HmiInterface".intCondition.Axis_08.Jog.intOut, workInterlockOK => "Unit1.Em5.ControlNodes".cm.Interlock.cathodeMainPnP2AxisX.permit.jogForward)
   END_RUNG
   RUNG wire#powerrail
      #"cathodeMainPnP2AxisX Jog_CCW"(Status := #unitStatus, HMI := "Unit1.Em5.HmiInterface".cmCathodeMainPnP2AxisX.commands.jogBackward, int1 :=, int2 :=, int3 :=, int4 :=, int5 :=, int6 :=, int7 :=, int8 :=, int9 :=, int10 :=, Bypass :=, intOut := "Unit1.Em5.HmiInterface".intCondition.Axis_08.Jog.intOut, workInterlockOK => "Unit1.Em5.ControlNodes".cm.Interlock.cathodeMainPnP2AxisX.permit.jogBackward)
   END_RUNG
   RUNG wire#powerrail
      I_Contact( #TRUE )
      Contact( "Unit1.Em5.ControlNodes".cm.Interlock.cathodeMainPnP2AxisX.permit.jogForward )
      Coil( "Unit1.Em5.ControlNodes".cmCathodeMainPnP2AxisX.commands.jogForward )
   END_RUNG
   RUNG wire#powerrail
      I_Contact( #TRUE )
      Contact( "Unit1.Em5.ControlNodes".cm.Interlock.cathodeMainPnP2AxisX.permit.jogBackward )
      Coil( "Unit1.Em5.ControlNodes".cmCathodeMainPnP2AxisX.commands.jogBackward )
   END_RUNG
   // the same network as SCL:
   #"cathodeMainPnP2AxisX Jog_CW"(Status := #unitStatus,   // "Jog.LER_Axis"
                           HMI := "Unit1.Em5.HmiInterface".cmCathodeMainPnP2AxisX.commands.jogForward,
                           intOut := "Unit1.Em5.HmiInterface".intCondition.Axis_08.Jog.intOut,
                           workInterlockOK => "Unit1.Em5.ControlNodes".cm.Interlock.cathodeMainPnP2AxisX.permit.jogForward);
   #"cathodeMainPnP2AxisX Jog_CCW"(Status := #unitStatus,   // "Jog.LER_Axis"
                           HMI := "Unit1.Em5.HmiInterface".cmCathodeMainPnP2AxisX.commands.jogBackward,
                           intOut := "Unit1.Em5.HmiInterface".intCondition.Axis_08.Jog.intOut,
                           workInterlockOK => "Unit1.Em5.ControlNodes".cm.Interlock.cathodeMainPnP2AxisX.permit.jogBackward);
   "Unit1.Em5.ControlNodes".cmCathodeMainPnP2AxisX.commands.jogForward := NOT #TRUE AND "Unit1.Em5.ControlNodes".cm.Interlock.cathodeMainPnP2AxisX.permit.jogForward;
   "Unit1.Em5.ControlNodes".cmCathodeMainPnP2AxisX.commands.jogBackward := NOT #TRUE AND "Unit1.Em5.ControlNodes".cm.Interlock.cathodeMainPnP2AxisX.permit.jogBackward;
END_REGION

REGION Network 132: CmCathodeMainPnP2AxisX Position Absolute Position0
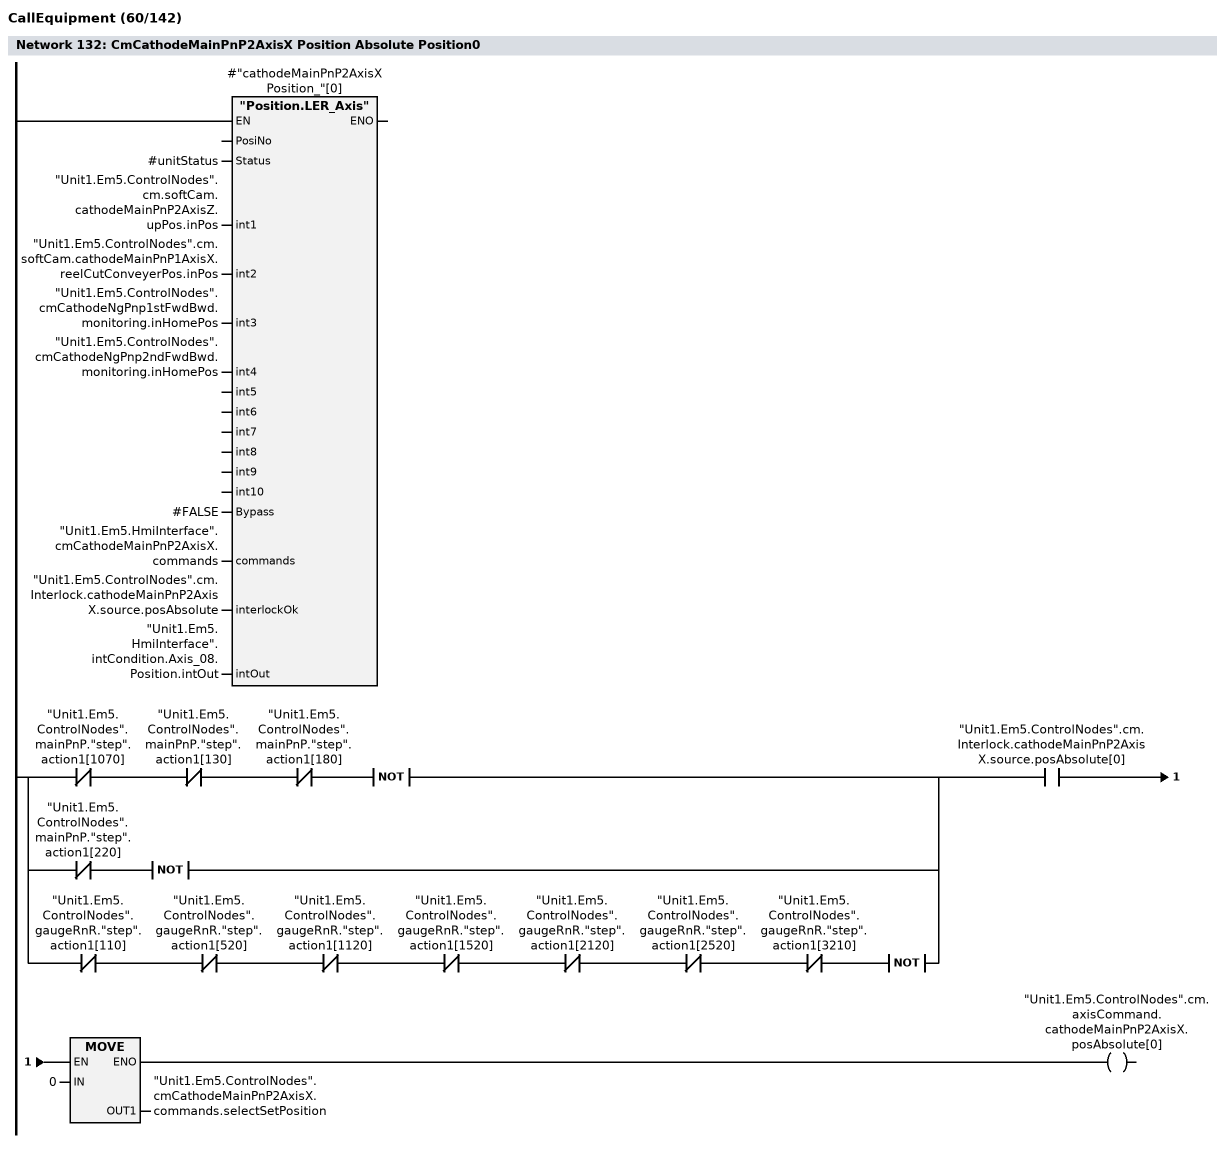
   RUNG wire#powerrail
      #"cathodeMainPnP2AxisX Position_"[0](PosiNo :=, Status := #unitStatus, int1 := "Unit1.Em5.ControlNodes".cm.softCam.cathodeMainPnP2AxisZ.upPos.inPos, int2 := "Unit1.Em5.ControlNodes".cm.softCam.cathodeMainPnP1AxisX.reelCutConveyerPos.inPos, int3 := "Unit1.Em5.ControlNodes".cmCathodeNgPnp1stFwdBwd.monitoring.inHomePos, int4 := "Unit1.Em5.ControlNodes".cmCathodeNgPnp2ndFwdBwd.monitoring.inHomePos, int5 :=, int6 :=, int7 :=, int8 :=, int9 :=, int10 :=, Bypass := #FALSE, commands := "Unit1.Em5.HmiInterface".cmCathodeMainPnP2AxisX.commands, interlockOk := "Unit1.Em5.ControlNodes".cm.Interlock.cathodeMainPnP2AxisX.source.posAbsolute, intOut := "Unit1.Em5.HmiInterface".intCondition.Axis_08.Position.intOut)
   END_RUNG
   RUNG wire#powerrail
      I_Contact( "Unit1.Em5.ControlNodes".mainPnP."step".action1[1070] )
      I_Contact( "Unit1.Em5.ControlNodes".mainPnP."step".action1[130] )
      I_Contact( "Unit1.Em5.ControlNodes".mainPnP."step".action1[180] )
      Not()
      wire#w1
      Contact( "Unit1.Em5.ControlNodes".cm.Interlock.cathodeMainPnP2AxisX.source.posAbsolute[0] )
      Move(in := 0, out1 => "Unit1.Em5.ControlNodes".cmCathodeMainPnP2AxisX.commands.selectSetPosition)
      Coil( "Unit1.Em5.ControlNodes".cm.axisCommand.cathodeMainPnP2AxisX.posAbsolute[0] )
   END_RUNG
   RUNG wire#powerrail
      I_Contact( "Unit1.Em5.ControlNodes".mainPnP."step".action1[220] )
      Not()
   END_RUNG wire#w1
   RUNG wire#powerrail
      I_Contact( "Unit1.Em5.ControlNodes".gaugeRnR."step".action1[110] )
      I_Contact( "Unit1.Em5.ControlNodes".gaugeRnR."step".action1[520] )
      I_Contact( "Unit1.Em5.ControlNodes".gaugeRnR."step".action1[1120] )
      I_Contact( "Unit1.Em5.ControlNodes".gaugeRnR."step".action1[1520] )
      I_Contact( "Unit1.Em5.ControlNodes".gaugeRnR."step".action1[2120] )
      I_Contact( "Unit1.Em5.ControlNodes".gaugeRnR."step".action1[2520] )
      I_Contact( "Unit1.Em5.ControlNodes".gaugeRnR."step".action1[3210] )
      Not()
   END_RUNG wire#w1
   // the same network as SCL:
   #"cathodeMainPnP2AxisX Position_"[0](Status := #unitStatus,   // "Position.LER_Axis"
                           int1 := "Unit1.Em5.ControlNodes".cm.softCam.cathodeMainPnP2AxisZ.upPos.inPos,
                           int2 := "Unit1.Em5.ControlNodes".cm.softCam.cathodeMainPnP1AxisX.reelCutConveyerPos.inPos,
                           int3 := "Unit1.Em5.ControlNodes".cmCathodeNgPnp1stFwdBwd.monitoring.inHomePos,
                           int4 := "Unit1.Em5.ControlNodes".cmCathodeNgPnp2ndFwdBwd.monitoring.inHomePos,
                           Bypass := #FALSE,
                           commands := "Unit1.Em5.HmiInterface".cmCathodeMainPnP2AxisX.commands,
                           interlockOk := "Unit1.Em5.ControlNodes".cm.Interlock.cathodeMainPnP2AxisX.source.posAbsolute,
                           intOut := "Unit1.Em5.HmiInterface".intCondition.Axis_08.Position.intOut);
   #_w1 := (NOT (NOT "Unit1.Em5.ControlNodes".mainPnP."step".action1[1070] AND NOT "Unit1.Em5.ControlNodes".mainPnP."step".action1[130] AND NOT "Unit1.Em5.ControlNodes".mainPnP."step".action1[180]) OR NOT (NOT "Unit1.Em5.ControlNodes".mainPnP."step".action1[220]) OR NOT (NOT "Unit1.Em5.ControlNodes".gaugeRnR."step".action1[110] AND NOT "Unit1.Em5.ControlNodes".gaugeRnR."step".action1[520] AND NOT "Unit1.Em5.ControlNodes".gaugeRnR."step".action1[1120] AND NOT "Unit1.Em5.ControlNodes".gaugeRnR."step".action1[1520] AND NOT "Unit1.Em5.ControlNodes".gaugeRnR."step".action1[2120] AND NOT "Unit1.Em5.ControlNodes".gaugeRnR."step".action1[2520] AND NOT "Unit1.Em5.ControlNodes".gaugeRnR."step".action1[3210])) AND "Unit1.Em5.ControlNodes".cm.Interlock.cathodeMainPnP2AxisX.source.posAbsolute[0];
   IF #_w1 THEN "Unit1.Em5.ControlNodes".cmCathodeMainPnP2AxisX.commands.selectSetPosition := 0; END_IF;
   "Unit1.Em5.ControlNodes".cm.axisCommand.cathodeMainPnP2AxisX.posAbsolute[0] := #_w1;
END_REGION

REGION Network 133: CmCathodeMainPnP2AxisX Position Absolute Position1
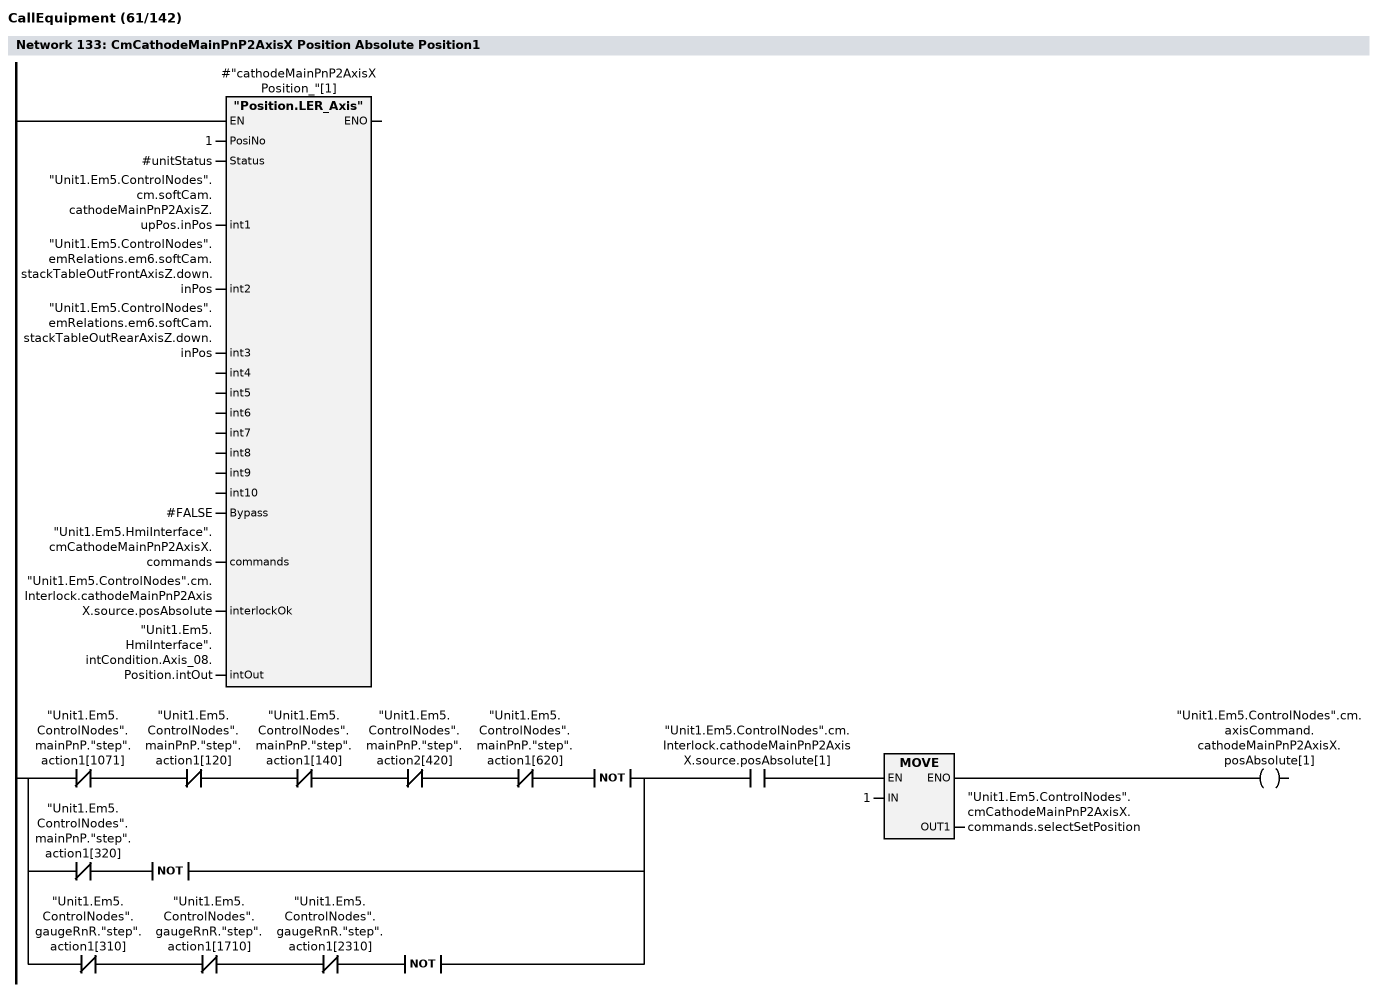
   RUNG wire#powerrail
      #"cathodeMainPnP2AxisX Position_"[1](PosiNo := 1, Status := #unitStatus, int1 := "Unit1.Em5.ControlNodes".cm.softCam.cathodeMainPnP2AxisZ.upPos.inPos, int2 := "Unit1.Em5.ControlNodes".emRelations.em6.softCam.stackTableOutFrontAxisZ.down.inPos, int3 := "Unit1.Em5.ControlNodes".emRelations.em6.softCam.stackTableOutRearAxisZ.down.inPos, int4 :=, int5 :=, int6 :=, int7 :=, int8 :=, int9 :=, int10 :=, Bypass := #FALSE, commands := "Unit1.Em5.HmiInterface".cmCathodeMainPnP2AxisX.commands, interlockOk := "Unit1.Em5.ControlNodes".cm.Interlock.cathodeMainPnP2AxisX.source.posAbsolute, intOut := "Unit1.Em5.HmiInterface".intCondition.Axis_08.Position.intOut)
   END_RUNG
   RUNG wire#powerrail
      I_Contact( "Unit1.Em5.ControlNodes".mainPnP."step".action1[1071] )
      I_Contact( "Unit1.Em5.ControlNodes".mainPnP."step".action1[120] )
      I_Contact( "Unit1.Em5.ControlNodes".mainPnP."step".action1[140] )
      I_Contact( "Unit1.Em5.ControlNodes".mainPnP."step".action2[420] )
      I_Contact( "Unit1.Em5.ControlNodes".mainPnP."step".action1[620] )
      Not()
      wire#w1
      Contact( "Unit1.Em5.ControlNodes".cm.Interlock.cathodeMainPnP2AxisX.source.posAbsolute[1] )
      Move(in := 1, out1 => "Unit1.Em5.ControlNodes".cmCathodeMainPnP2AxisX.commands.selectSetPosition)
      Coil( "Unit1.Em5.ControlNodes".cm.axisCommand.cathodeMainPnP2AxisX.posAbsolute[1] )
   END_RUNG
   RUNG wire#powerrail
      I_Contact( "Unit1.Em5.ControlNodes".mainPnP."step".action1[320] )
      Not()
   END_RUNG wire#w1
   RUNG wire#powerrail
      I_Contact( "Unit1.Em5.ControlNodes".gaugeRnR."step".action1[310] )
      I_Contact( "Unit1.Em5.ControlNodes".gaugeRnR."step".action1[1710] )
      I_Contact( "Unit1.Em5.ControlNodes".gaugeRnR."step".action1[2310] )
      Not()
   END_RUNG wire#w1
   // the same network as SCL:
   #"cathodeMainPnP2AxisX Position_"[1](PosiNo := 1,   // "Position.LER_Axis"
                           Status := #unitStatus,
                           int1 := "Unit1.Em5.ControlNodes".cm.softCam.cathodeMainPnP2AxisZ.upPos.inPos,
                           int2 := "Unit1.Em5.ControlNodes".emRelations.em6.softCam.stackTableOutFrontAxisZ.down.inPos,
                           int3 := "Unit1.Em5.ControlNodes".emRelations.em6.softCam.stackTableOutRearAxisZ.down.inPos,
                           Bypass := #FALSE,
                           commands := "Unit1.Em5.HmiInterface".cmCathodeMainPnP2AxisX.commands,
                           interlockOk := "Unit1.Em5.ControlNodes".cm.Interlock.cathodeMainPnP2AxisX.source.posAbsolute,
                           intOut := "Unit1.Em5.HmiInterface".intCondition.Axis_08.Position.intOut);
   #_w1 := (NOT (NOT "Unit1.Em5.ControlNodes".mainPnP."step".action1[1071] AND NOT "Unit1.Em5.ControlNodes".mainPnP."step".action1[120] AND NOT "Unit1.Em5.ControlNodes".mainPnP."step".action1[140] AND NOT "Unit1.Em5.ControlNodes".mainPnP."step".action2[420] AND NOT "Unit1.Em5.ControlNodes".mainPnP."step".action1[620]) OR NOT (NOT "Unit1.Em5.ControlNodes".mainPnP."step".action1[320]) OR NOT (NOT "Unit1.Em5.ControlNodes".gaugeRnR."step".action1[310] AND NOT "Unit1.Em5.ControlNodes".gaugeRnR."step".action1[1710] AND NOT "Unit1.Em5.ControlNodes".gaugeRnR."step".action1[2310])) AND "Unit1.Em5.ControlNodes".cm.Interlock.cathodeMainPnP2AxisX.source.posAbsolute[1];
   IF #_w1 THEN "Unit1.Em5.ControlNodes".cmCathodeMainPnP2AxisX.commands.selectSetPosition := 1; END_IF;
   "Unit1.Em5.ControlNodes".cm.axisCommand.cathodeMainPnP2AxisX.posAbsolute[1] := #_w1;
END_REGION

REGION Network 134: CmCathodeMainPnP2AxisX Position Absolute Position2
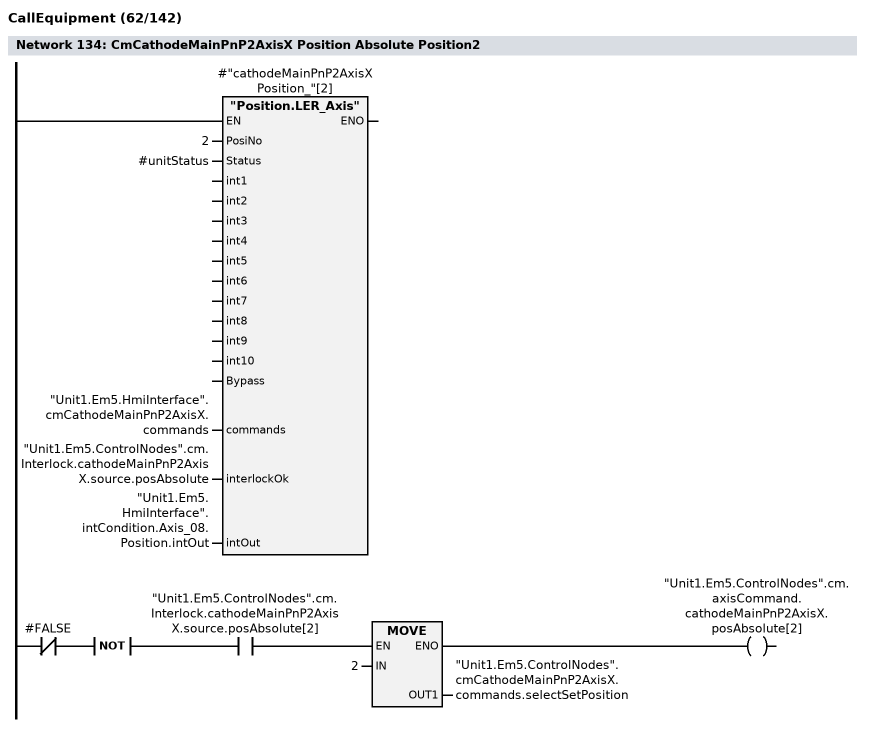
   RUNG wire#powerrail
      #"cathodeMainPnP2AxisX Position_"[2](PosiNo := 2, Status := #unitStatus, int1 :=, int2 :=, int3 :=, int4 :=, int5 :=, int6 :=, int7 :=, int8 :=, int9 :=, int10 :=, Bypass :=, commands := "Unit1.Em5.HmiInterface".cmCathodeMainPnP2AxisX.commands, interlockOk := "Unit1.Em5.ControlNodes".cm.Interlock.cathodeMainPnP2AxisX.source.posAbsolute, intOut := "Unit1.Em5.HmiInterface".intCondition.Axis_08.Position.intOut)
   END_RUNG
   RUNG wire#powerrail
      I_Contact( #FALSE )
      Not()
      Contact( "Unit1.Em5.ControlNodes".cm.Interlock.cathodeMainPnP2AxisX.source.posAbsolute[2] )
      Move(in := 2, out1 => "Unit1.Em5.ControlNodes".cmCathodeMainPnP2AxisX.commands.selectSetPosition)
      Coil( "Unit1.Em5.ControlNodes".cm.axisCommand.cathodeMainPnP2AxisX.posAbsolute[2] )
   END_RUNG
   // the same network as SCL:
   #"cathodeMainPnP2AxisX Position_"[2](PosiNo := 2,   // "Position.LER_Axis"
                           Status := #unitStatus,
                           commands := "Unit1.Em5.HmiInterface".cmCathodeMainPnP2AxisX.commands,
                           interlockOk := "Unit1.Em5.ControlNodes".cm.Interlock.cathodeMainPnP2AxisX.source.posAbsolute,
                           intOut := "Unit1.Em5.HmiInterface".intCondition.Axis_08.Position.intOut);
   #_w1 := NOT (NOT #FALSE) AND "Unit1.Em5.ControlNodes".cm.Interlock.cathodeMainPnP2AxisX.source.posAbsolute[2];
   IF #_w1 THEN "Unit1.Em5.ControlNodes".cmCathodeMainPnP2AxisX.commands.selectSetPosition := 2; END_IF;
   "Unit1.Em5.ControlNodes".cm.axisCommand.cathodeMainPnP2AxisX.posAbsolute[2] := #_w1;
END_REGION

REGION Network 135: CmCathodeMainPnP2AxisX Position Absolute Position3
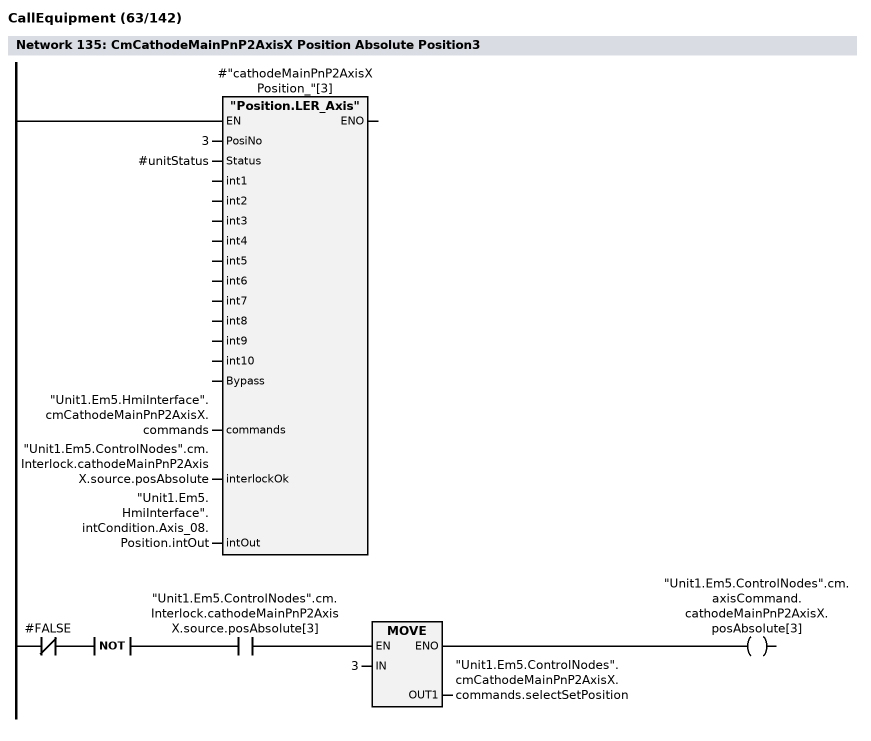
   RUNG wire#powerrail
      #"cathodeMainPnP2AxisX Position_"[3](PosiNo := 3, Status := #unitStatus, int1 :=, int2 :=, int3 :=, int4 :=, int5 :=, int6 :=, int7 :=, int8 :=, int9 :=, int10 :=, Bypass :=, commands := "Unit1.Em5.HmiInterface".cmCathodeMainPnP2AxisX.commands, interlockOk := "Unit1.Em5.ControlNodes".cm.Interlock.cathodeMainPnP2AxisX.source.posAbsolute, intOut := "Unit1.Em5.HmiInterface".intCondition.Axis_08.Position.intOut)
   END_RUNG
   RUNG wire#powerrail
      I_Contact( #FALSE )
      Not()
      Contact( "Unit1.Em5.ControlNodes".cm.Interlock.cathodeMainPnP2AxisX.source.posAbsolute[3] )
      Move(in := 3, out1 => "Unit1.Em5.ControlNodes".cmCathodeMainPnP2AxisX.commands.selectSetPosition)
      Coil( "Unit1.Em5.ControlNodes".cm.axisCommand.cathodeMainPnP2AxisX.posAbsolute[3] )
   END_RUNG
   // the same network as SCL:
   #"cathodeMainPnP2AxisX Position_"[3](PosiNo := 3,   // "Position.LER_Axis"
                           Status := #unitStatus,
                           commands := "Unit1.Em5.HmiInterface".cmCathodeMainPnP2AxisX.commands,
                           interlockOk := "Unit1.Em5.ControlNodes".cm.Interlock.cathodeMainPnP2AxisX.source.posAbsolute,
                           intOut := "Unit1.Em5.HmiInterface".intCondition.Axis_08.Position.intOut);
   #_w1 := NOT (NOT #FALSE) AND "Unit1.Em5.ControlNodes".cm.Interlock.cathodeMainPnP2AxisX.source.posAbsolute[3];
   IF #_w1 THEN "Unit1.Em5.ControlNodes".cmCathodeMainPnP2AxisX.commands.selectSetPosition := 3; END_IF;
   "Unit1.Em5.ControlNodes".cm.axisCommand.cathodeMainPnP2AxisX.posAbsolute[3] := #_w1;
END_REGION

REGION Network 136: CmCathodeMainPnP2AxisX Position Absolute Position4
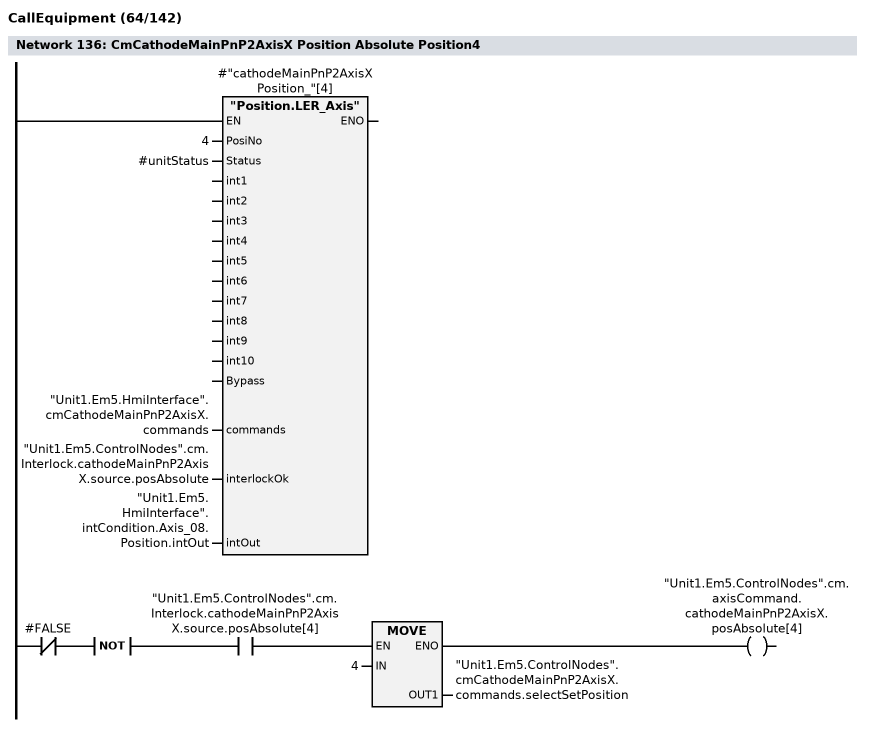
   RUNG wire#powerrail
      #"cathodeMainPnP2AxisX Position_"[4](PosiNo := 4, Status := #unitStatus, int1 :=, int2 :=, int3 :=, int4 :=, int5 :=, int6 :=, int7 :=, int8 :=, int9 :=, int10 :=, Bypass :=, commands := "Unit1.Em5.HmiInterface".cmCathodeMainPnP2AxisX.commands, interlockOk := "Unit1.Em5.ControlNodes".cm.Interlock.cathodeMainPnP2AxisX.source.posAbsolute, intOut := "Unit1.Em5.HmiInterface".intCondition.Axis_08.Position.intOut)
   END_RUNG
   RUNG wire#powerrail
      I_Contact( #FALSE )
      Not()
      Contact( "Unit1.Em5.ControlNodes".cm.Interlock.cathodeMainPnP2AxisX.source.posAbsolute[4] )
      Move(in := 4, out1 => "Unit1.Em5.ControlNodes".cmCathodeMainPnP2AxisX.commands.selectSetPosition)
      Coil( "Unit1.Em5.ControlNodes".cm.axisCommand.cathodeMainPnP2AxisX.posAbsolute[4] )
   END_RUNG
   // the same network as SCL:
   #"cathodeMainPnP2AxisX Position_"[4](PosiNo := 4,   // "Position.LER_Axis"
                           Status := #unitStatus,
                           commands := "Unit1.Em5.HmiInterface".cmCathodeMainPnP2AxisX.commands,
                           interlockOk := "Unit1.Em5.ControlNodes".cm.Interlock.cathodeMainPnP2AxisX.source.posAbsolute,
                           intOut := "Unit1.Em5.HmiInterface".intCondition.Axis_08.Position.intOut);
   #_w1 := NOT (NOT #FALSE) AND "Unit1.Em5.ControlNodes".cm.Interlock.cathodeMainPnP2AxisX.source.posAbsolute[4];
   IF #_w1 THEN "Unit1.Em5.ControlNodes".cmCathodeMainPnP2AxisX.commands.selectSetPosition := 4; END_IF;
   "Unit1.Em5.ControlNodes".cm.axisCommand.cathodeMainPnP2AxisX.posAbsolute[4] := #_w1;
END_REGION

REGION Network 137: CmCathodeMainPnP2AxisX Position Absolute Position5
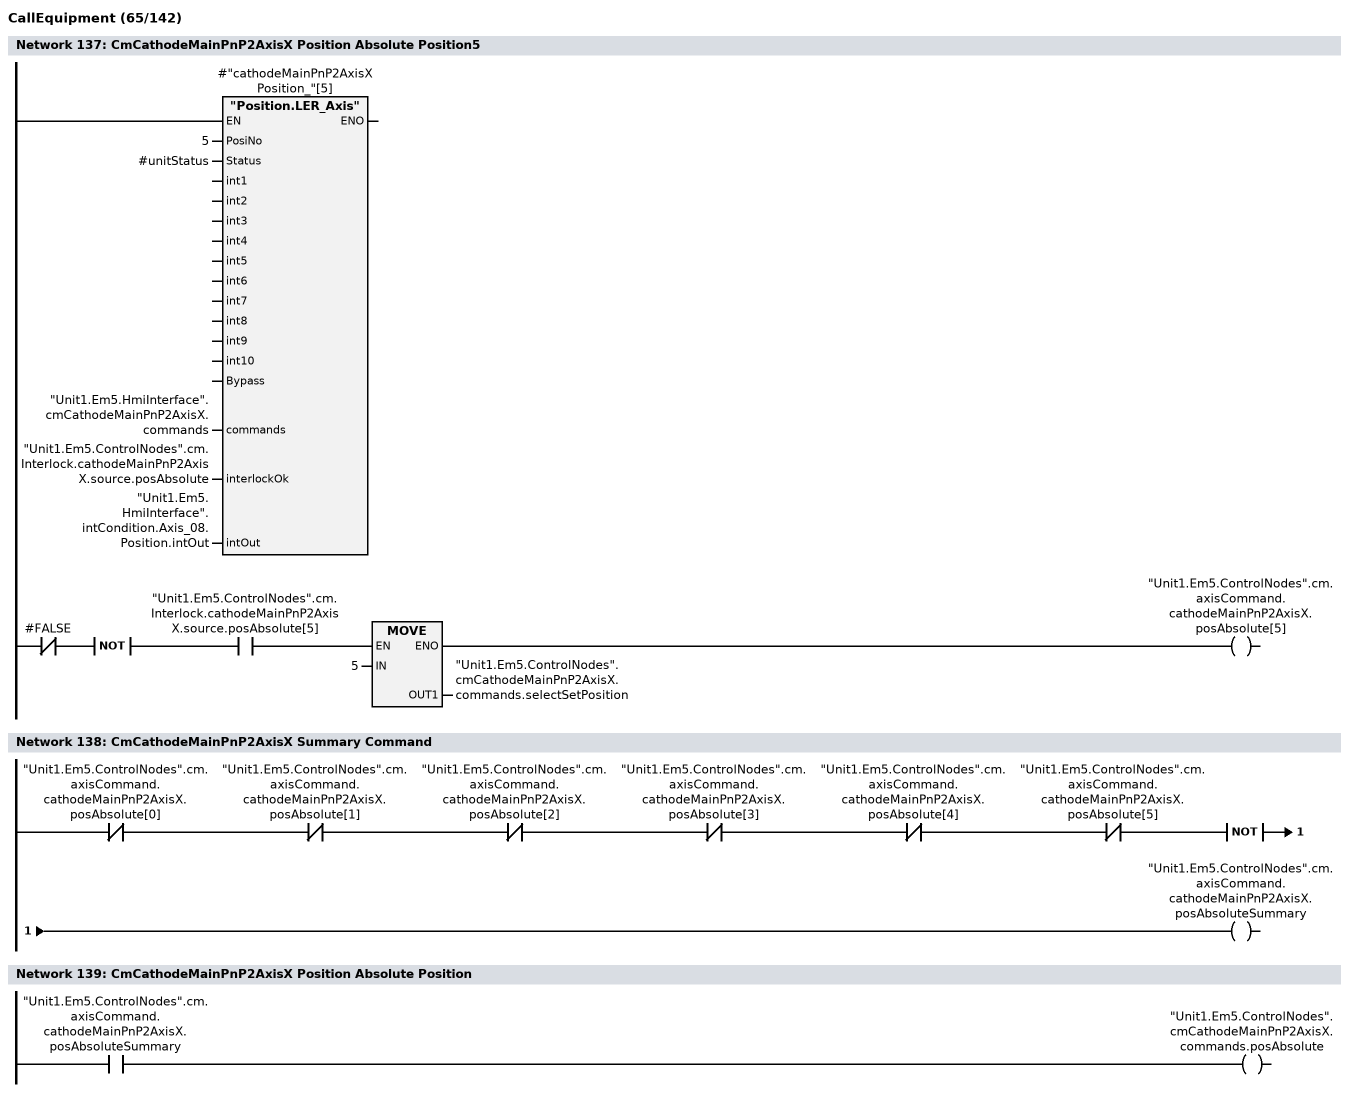
   RUNG wire#powerrail
      #"cathodeMainPnP2AxisX Position_"[5](PosiNo := 5, Status := #unitStatus, int1 :=, int2 :=, int3 :=, int4 :=, int5 :=, int6 :=, int7 :=, int8 :=, int9 :=, int10 :=, Bypass :=, commands := "Unit1.Em5.HmiInterface".cmCathodeMainPnP2AxisX.commands, interlockOk := "Unit1.Em5.ControlNodes".cm.Interlock.cathodeMainPnP2AxisX.source.posAbsolute, intOut := "Unit1.Em5.HmiInterface".intCondition.Axis_08.Position.intOut)
   END_RUNG
   RUNG wire#powerrail
      I_Contact( #FALSE )
      Not()
      Contact( "Unit1.Em5.ControlNodes".cm.Interlock.cathodeMainPnP2AxisX.source.posAbsolute[5] )
      Move(in := 5, out1 => "Unit1.Em5.ControlNodes".cmCathodeMainPnP2AxisX.commands.selectSetPosition)
      Coil( "Unit1.Em5.ControlNodes".cm.axisCommand.cathodeMainPnP2AxisX.posAbsolute[5] )
   END_RUNG
   // the same network as SCL:
   #"cathodeMainPnP2AxisX Position_"[5](PosiNo := 5,   // "Position.LER_Axis"
                           Status := #unitStatus,
                           commands := "Unit1.Em5.HmiInterface".cmCathodeMainPnP2AxisX.commands,
                           interlockOk := "Unit1.Em5.ControlNodes".cm.Interlock.cathodeMainPnP2AxisX.source.posAbsolute,
                           intOut := "Unit1.Em5.HmiInterface".intCondition.Axis_08.Position.intOut);
   #_w1 := NOT (NOT #FALSE) AND "Unit1.Em5.ControlNodes".cm.Interlock.cathodeMainPnP2AxisX.source.posAbsolute[5];
   IF #_w1 THEN "Unit1.Em5.ControlNodes".cmCathodeMainPnP2AxisX.commands.selectSetPosition := 5; END_IF;
   "Unit1.Em5.ControlNodes".cm.axisCommand.cathodeMainPnP2AxisX.posAbsolute[5] := #_w1;
END_REGION

REGION Network 138: CmCathodeMainPnP2AxisX Summary Command
   RUNG wire#powerrail
      I_Contact( "Unit1.Em5.ControlNodes".cm.axisCommand.cathodeMainPnP2AxisX.posAbsolute[0] )
      I_Contact( "Unit1.Em5.ControlNodes".cm.axisCommand.cathodeMainPnP2AxisX.posAbsolute[1] )
      I_Contact( "Unit1.Em5.ControlNodes".cm.axisCommand.cathodeMainPnP2AxisX.posAbsolute[2] )
      I_Contact( "Unit1.Em5.ControlNodes".cm.axisCommand.cathodeMainPnP2AxisX.posAbsolute[3] )
      I_Contact( "Unit1.Em5.ControlNodes".cm.axisCommand.cathodeMainPnP2AxisX.posAbsolute[4] )
      I_Contact( "Unit1.Em5.ControlNodes".cm.axisCommand.cathodeMainPnP2AxisX.posAbsolute[5] )
      Not()
      Coil( "Unit1.Em5.ControlNodes".cm.axisCommand.cathodeMainPnP2AxisX.posAbsoluteSummary )
   END_RUNG
   // the same network as SCL:
   "Unit1.Em5.ControlNodes".cm.axisCommand.cathodeMainPnP2AxisX.posAbsoluteSummary := NOT (NOT "Unit1.Em5.ControlNodes".cm.axisCommand.cathodeMainPnP2AxisX.posAbsolute[0] AND NOT "Unit1.Em5.ControlNodes".cm.axisCommand.cathodeMainPnP2AxisX.posAbsolute[1] AND NOT "Unit1.Em5.ControlNodes".cm.axisCommand.cathodeMainPnP2AxisX.posAbsolute[2] AND NOT "Unit1.Em5.ControlNodes".cm.axisCommand.cathodeMainPnP2AxisX.posAbsolute[3] AND NOT "Unit1.Em5.ControlNodes".cm.axisCommand.cathodeMainPnP2AxisX.posAbsolute[4] AND NOT "Unit1.Em5.ControlNodes".cm.axisCommand.cathodeMainPnP2AxisX.posAbsolute[5]);
END_REGION

REGION Network 139: CmCathodeMainPnP2AxisX Position Absolute Position
   RUNG wire#powerrail
      Contact( "Unit1.Em5.ControlNodes".cm.axisCommand.cathodeMainPnP2AxisX.posAbsoluteSummary )
      Coil( "Unit1.Em5.ControlNodes".cmCathodeMainPnP2AxisX.commands.posAbsolute )
   END_RUNG
   // the same network as SCL:
   "Unit1.Em5.ControlNodes".cmCathodeMainPnP2AxisX.commands.posAbsolute := "Unit1.Em5.ControlNodes".cm.axisCommand.cathodeMainPnP2AxisX.posAbsoluteSummary;
END_REGION

REGION Network 140: CmCathodeMainPnP2AxisX Interlock Summary
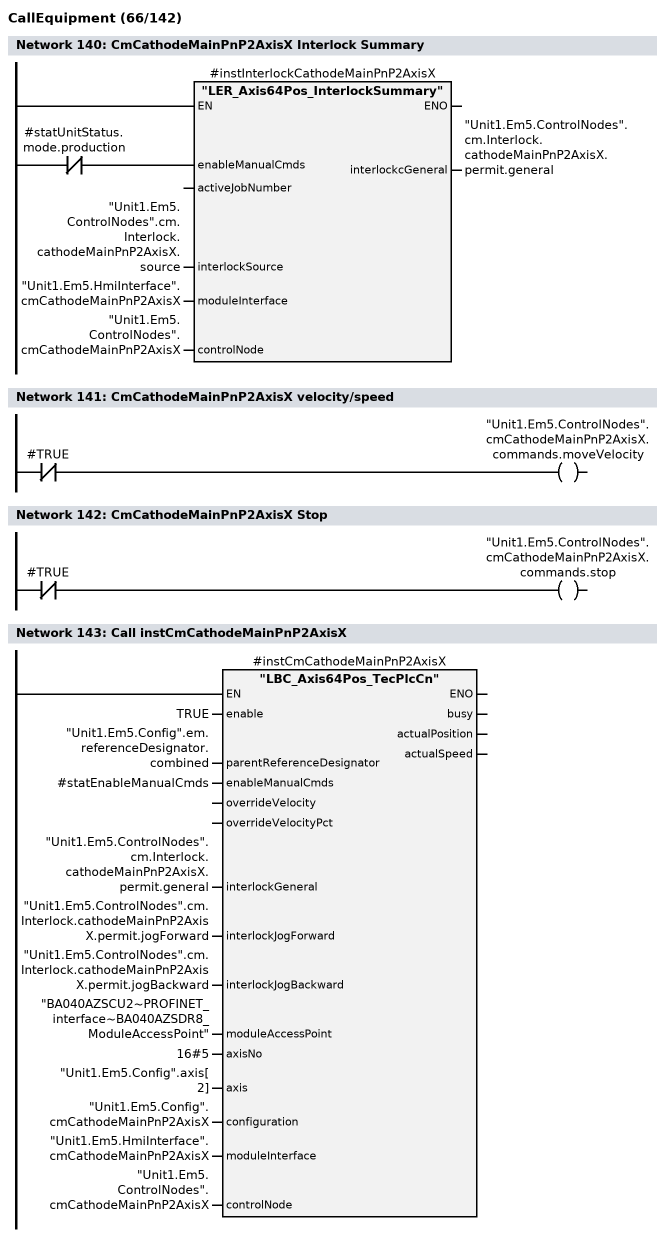
   RUNG wire#powerrail
      #instInterlockCathodeMainPnP2AxisX(enableManualCmds := wire#w1, activeJobNumber :=, interlockSource := "Unit1.Em5.ControlNodes".cm.Interlock.cathodeMainPnP2AxisX.source, moduleInterface := "Unit1.Em5.HmiInterface".cmCathodeMainPnP2AxisX, controlNode := "Unit1.Em5.ControlNodes".cmCathodeMainPnP2AxisX, interlockcGeneral => "Unit1.Em5.ControlNodes".cm.Interlock.cathodeMainPnP2AxisX.permit.general)
   END_RUNG
   RUNG wire#powerrail
      I_Contact( #statUnitStatus.mode.production )
   END_RUNG wire#w1
   // the same network as SCL:
   #instInterlockCathodeMainPnP2AxisX(enableManualCmds := NOT #statUnitStatus.mode.production,   // "LER_Axis64Pos_InterlockSummary"
                           interlockSource := "Unit1.Em5.ControlNodes".cm.Interlock.cathodeMainPnP2AxisX.source,
                           moduleInterface := "Unit1.Em5.HmiInterface".cmCathodeMainPnP2AxisX,
                           controlNode := "Unit1.Em5.ControlNodes".cmCathodeMainPnP2AxisX,
                           interlockcGeneral => "Unit1.Em5.ControlNodes".cm.Interlock.cathodeMainPnP2AxisX.permit.general);
END_REGION

REGION Network 141: CmCathodeMainPnP2AxisX velocity/speed
   RUNG wire#powerrail
      I_Contact( #TRUE )
      Coil( "Unit1.Em5.ControlNodes".cmCathodeMainPnP2AxisX.commands.moveVelocity )
   END_RUNG
   // the same network as SCL:
   "Unit1.Em5.ControlNodes".cmCathodeMainPnP2AxisX.commands.moveVelocity := NOT #TRUE;
END_REGION

REGION Network 142: CmCathodeMainPnP2AxisX Stop
   RUNG wire#powerrail
      I_Contact( #TRUE )
      Coil( "Unit1.Em5.ControlNodes".cmCathodeMainPnP2AxisX.commands.stop )
   END_RUNG
   // the same network as SCL:
   "Unit1.Em5.ControlNodes".cmCathodeMainPnP2AxisX.commands.stop := NOT #TRUE;
END_REGION

REGION Network 143: Call instCmCathodeMainPnP2AxisX
   RUNG wire#powerrail
      #instCmCathodeMainPnP2AxisX(enable := TRUE, parentReferenceDesignator := "Unit1.Em5.Config".em.referenceDesignator.combined, enableManualCmds := #statEnableManualCmds, overrideVelocity :=, overrideVelocityPct :=, interlockGeneral := "Unit1.Em5.ControlNodes".cm.Interlock.cathodeMainPnP2AxisX.permit.general, interlockJogForward := "Unit1.Em5.ControlNodes".cm.Interlock.cathodeMainPnP2AxisX.permit.jogForward, interlockJogBackward := "Unit1.Em5.ControlNodes".cm.Interlock.cathodeMainPnP2AxisX.permit.jogBackward, moduleAccessPoint := "BA040AZSCU2~PROFINET_interface~BA040AZSDR8_ModuleAccessPoint", axisNo := 16#5, axis := "Unit1.Em5.Config".axis[2], configuration := "Unit1.Em5.Config".cmCathodeMainPnP2AxisX, moduleInterface := "Unit1.Em5.HmiInterface".cmCathodeMainPnP2AxisX, controlNode := "Unit1.Em5.ControlNodes".cmCathodeMainPnP2AxisX, busy =>, actualPosition =>, actualSpeed =>)
   END_RUNG
   // the same network as SCL:
   #instCmCathodeMainPnP2AxisX(enable := TRUE,   // "LBC_Axis64Pos_TecPlcCn"
                           parentReferenceDesignator := "Unit1.Em5.Config".em.referenceDesignator.combined,
                           enableManualCmds := #statEnableManualCmds,
                           interlockGeneral := "Unit1.Em5.ControlNodes".cm.Interlock.cathodeMainPnP2AxisX.permit.general,
                           interlockJogForward := "Unit1.Em5.ControlNodes".cm.Interlock.cathodeMainPnP2AxisX.permit.jogForward,
                           interlockJogBackward := "Unit1.Em5.ControlNodes".cm.Interlock.cathodeMainPnP2AxisX.permit.jogBackward,
                           moduleAccessPoint := "BA040AZSCU2~PROFINET_interface~BA040AZSDR8_ModuleAccessPoint",
                           axisNo := 16#5,
                           axis := "Unit1.Em5.Config".axis[2],
                           configuration := "Unit1.Em5.Config".cmCathodeMainPnP2AxisX,
                           moduleInterface := "Unit1.Em5.HmiInterface".cmCathodeMainPnP2AxisX,
                           controlNode := "Unit1.Em5.ControlNodes".cmCathodeMainPnP2AxisX);
END_REGION

REGION Network 144: CmCathodeMainPnP2AxisX SoftCam
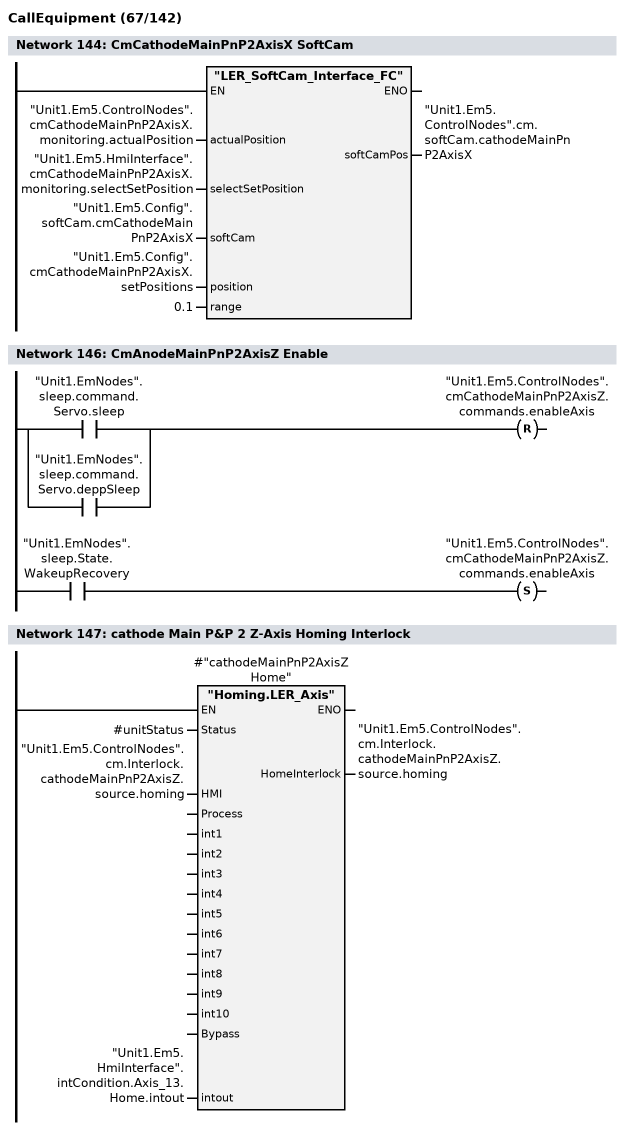
   RUNG wire#powerrail
      "LER_SoftCam_Interface_FC"(actualPosition := "Unit1.Em5.ControlNodes".cmCathodeMainPnP2AxisX.monitoring.actualPosition, selectSetPosition := "Unit1.Em5.HmiInterface".cmCathodeMainPnP2AxisX.monitoring.selectSetPosition, softCam := "Unit1.Em5.Config".softCam.cmCathodeMainPnP2AxisX, position := "Unit1.Em5.Config".cmCathodeMainPnP2AxisX.setPositions, range := 0.1, softCamPos => "Unit1.Em5.ControlNodes".cm.softCam.cathodeMainPnP2AxisX)
   END_RUNG
   // the same network as SCL:
   "LER_SoftCam_Interface_FC"(actualPosition := "Unit1.Em5.ControlNodes".cmCathodeMainPnP2AxisX.monitoring.actualPosition,
                           selectSetPosition := "Unit1.Em5.HmiInterface".cmCathodeMainPnP2AxisX.monitoring.selectSetPosition,
                           softCam := "Unit1.Em5.Config".softCam.cmCathodeMainPnP2AxisX,
                           position := "Unit1.Em5.Config".cmCathodeMainPnP2AxisX.setPositions,
                           range := 0.1,
                           softCamPos => "Unit1.Em5.ControlNodes".cm.softCam.cathodeMainPnP2AxisX);
END_REGION

REGION Network 146: CmAnodeMainPnP2AxisZ Enable
   RUNG wire#powerrail
      Contact( "Unit1.EmNodes".sleep.command.Servo.sleep )
      wire#w1
      R_Coil( "Unit1.Em5.ControlNodes".cmCathodeMainPnP2AxisZ.commands.enableAxis )
   END_RUNG
   RUNG wire#powerrail
      Contact( "Unit1.EmNodes".sleep.command.Servo.deppSleep )
   END_RUNG wire#w1
   RUNG wire#powerrail
      Contact( "Unit1.EmNodes".sleep.State.WakeupRecovery )
      S_Coil( "Unit1.Em5.ControlNodes".cmCathodeMainPnP2AxisZ.commands.enableAxis )
   END_RUNG
   // the same network as SCL:
   IF "Unit1.EmNodes".sleep.command.Servo.sleep OR "Unit1.EmNodes".sleep.command.Servo.deppSleep THEN
       "Unit1.Em5.ControlNodes".cmCathodeMainPnP2AxisZ.commands.enableAxis := FALSE;
   END_IF;
   IF "Unit1.EmNodes".sleep.State.WakeupRecovery THEN
       "Unit1.Em5.ControlNodes".cmCathodeMainPnP2AxisZ.commands.enableAxis := TRUE;
   END_IF;
END_REGION

REGION Network 147: cathode Main P&P 2 Z-Axis Homing Interlock
   RUNG wire#powerrail
      #"cathodeMainPnP2AxisZ Home"(Status := #unitStatus, HMI := "Unit1.Em5.ControlNodes".cm.Interlock.cathodeMainPnP2AxisZ.source.homing, Process :=, int1 :=, int2 :=, int3 :=, int4 :=, int5 :=, int6 :=, int7 :=, int8 :=, int9 :=, int10 :=, Bypass :=, intout := "Unit1.Em5.HmiInterface".intCondition.Axis_13.Home.intout, HomeInterlock => "Unit1.Em5.ControlNodes".cm.Interlock.cathodeMainPnP2AxisZ.source.homing)
   END_RUNG
   // the same network as SCL:
   #"cathodeMainPnP2AxisZ Home"(Status := #unitStatus,   // "Homing.LER_Axis"
                           HMI := "Unit1.Em5.ControlNodes".cm.Interlock.cathodeMainPnP2AxisZ.source.homing,
                           intout := "Unit1.Em5.HmiInterface".intCondition.Axis_13.Home.intout,
                           HomeInterlock => "Unit1.Em5.ControlNodes".cm.Interlock.cathodeMainPnP2AxisZ.source.homing);
END_REGION

REGION Network 148: CmCathodeMainPnP2AxisZ Position Absolute Jog
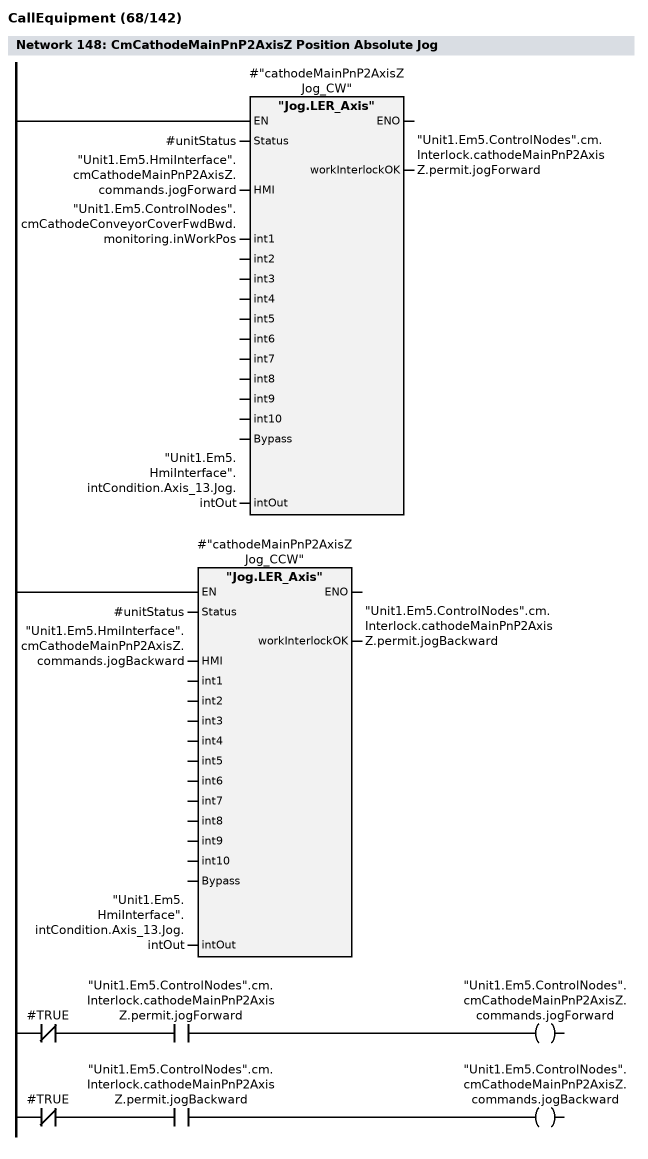
   RUNG wire#powerrail
      #"cathodeMainPnP2AxisZ Jog_CW"(Status := #unitStatus, HMI := "Unit1.Em5.HmiInterface".cmCathodeMainPnP2AxisZ.commands.jogForward, int1 := "Unit1.Em5.ControlNodes".cmCathodeConveyorCoverFwdBwd.monitoring.inWorkPos, int2 :=, int3 :=, int4 :=, int5 :=, int6 :=, int7 :=, int8 :=, int9 :=, int10 :=, Bypass :=, intOut := "Unit1.Em5.HmiInterface".intCondition.Axis_13.Jog.intOut, workInterlockOK => "Unit1.Em5.ControlNodes".cm.Interlock.cathodeMainPnP2AxisZ.permit.jogForward)
   END_RUNG
   RUNG wire#powerrail
      #"cathodeMainPnP2AxisZ Jog_CCW"(Status := #unitStatus, HMI := "Unit1.Em5.HmiInterface".cmCathodeMainPnP2AxisZ.commands.jogBackward, int1 :=, int2 :=, int3 :=, int4 :=, int5 :=, int6 :=, int7 :=, int8 :=, int9 :=, int10 :=, Bypass :=, intOut := "Unit1.Em5.HmiInterface".intCondition.Axis_13.Jog.intOut, workInterlockOK => "Unit1.Em5.ControlNodes".cm.Interlock.cathodeMainPnP2AxisZ.permit.jogBackward)
   END_RUNG
   RUNG wire#powerrail
      I_Contact( #TRUE )
      Contact( "Unit1.Em5.ControlNodes".cm.Interlock.cathodeMainPnP2AxisZ.permit.jogForward )
      Coil( "Unit1.Em5.ControlNodes".cmCathodeMainPnP2AxisZ.commands.jogForward )
   END_RUNG
   RUNG wire#powerrail
      I_Contact( #TRUE )
      Contact( "Unit1.Em5.ControlNodes".cm.Interlock.cathodeMainPnP2AxisZ.permit.jogBackward )
      Coil( "Unit1.Em5.ControlNodes".cmCathodeMainPnP2AxisZ.commands.jogBackward )
   END_RUNG
   // the same network as SCL:
   #"cathodeMainPnP2AxisZ Jog_CW"(Status := #unitStatus,   // "Jog.LER_Axis"
                           HMI := "Unit1.Em5.HmiInterface".cmCathodeMainPnP2AxisZ.commands.jogForward,
                           int1 := "Unit1.Em5.ControlNodes".cmCathodeConveyorCoverFwdBwd.monitoring.inWorkPos,
                           intOut := "Unit1.Em5.HmiInterface".intCondition.Axis_13.Jog.intOut,
                           workInterlockOK => "Unit1.Em5.ControlNodes".cm.Interlock.cathodeMainPnP2AxisZ.permit.jogForward);
   #"cathodeMainPnP2AxisZ Jog_CCW"(Status := #unitStatus,   // "Jog.LER_Axis"
                           HMI := "Unit1.Em5.HmiInterface".cmCathodeMainPnP2AxisZ.commands.jogBackward,
                           intOut := "Unit1.Em5.HmiInterface".intCondition.Axis_13.Jog.intOut,
                           workInterlockOK => "Unit1.Em5.ControlNodes".cm.Interlock.cathodeMainPnP2AxisZ.permit.jogBackward);
   "Unit1.Em5.ControlNodes".cmCathodeMainPnP2AxisZ.commands.jogForward := NOT #TRUE AND "Unit1.Em5.ControlNodes".cm.Interlock.cathodeMainPnP2AxisZ.permit.jogForward;
   "Unit1.Em5.ControlNodes".cmCathodeMainPnP2AxisZ.commands.jogBackward := NOT #TRUE AND "Unit1.Em5.ControlNodes".cm.Interlock.cathodeMainPnP2AxisZ.permit.jogBackward;
END_REGION

REGION Network 149: CmCathodeMainPnP2AxisZ Position Absolute Position0
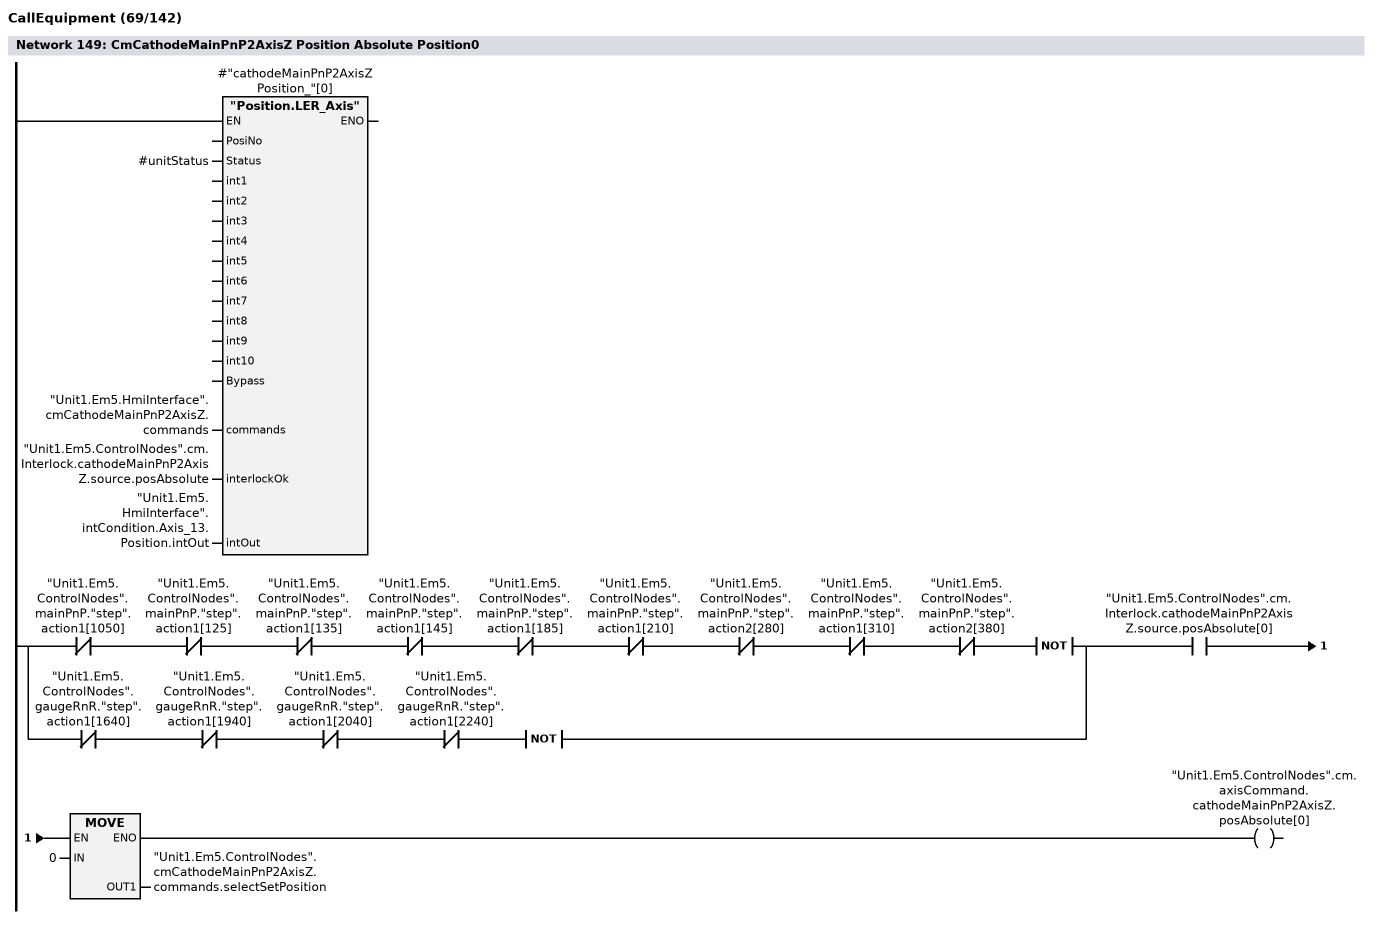
   RUNG wire#powerrail
      #"cathodeMainPnP2AxisZ Position_"[0](PosiNo :=, Status := #unitStatus, int1 :=, int2 :=, int3 :=, int4 :=, int5 :=, int6 :=, int7 :=, int8 :=, int9 :=, int10 :=, Bypass :=, commands := "Unit1.Em5.HmiInterface".cmCathodeMainPnP2AxisZ.commands, interlockOk := "Unit1.Em5.ControlNodes".cm.Interlock.cathodeMainPnP2AxisZ.source.posAbsolute, intOut := "Unit1.Em5.HmiInterface".intCondition.Axis_13.Position.intOut)
   END_RUNG
   RUNG wire#powerrail
      I_Contact( "Unit1.Em5.ControlNodes".mainPnP."step".action1[1050] )
      I_Contact( "Unit1.Em5.ControlNodes".mainPnP."step".action1[125] )
      I_Contact( "Unit1.Em5.ControlNodes".mainPnP."step".action1[135] )
      I_Contact( "Unit1.Em5.ControlNodes".mainPnP."step".action1[145] )
      I_Contact( "Unit1.Em5.ControlNodes".mainPnP."step".action1[185] )
      I_Contact( "Unit1.Em5.ControlNodes".mainPnP."step".action1[210] )
      I_Contact( "Unit1.Em5.ControlNodes".mainPnP."step".action2[280] )
      I_Contact( "Unit1.Em5.ControlNodes".mainPnP."step".action1[310] )
      I_Contact( "Unit1.Em5.ControlNodes".mainPnP."step".action2[380] )
      Not()
      wire#w1
      Contact( "Unit1.Em5.ControlNodes".cm.Interlock.cathodeMainPnP2AxisZ.source.posAbsolute[0] )
      Move(in := 0, out1 => "Unit1.Em5.ControlNodes".cmCathodeMainPnP2AxisZ.commands.selectSetPosition)
      Coil( "Unit1.Em5.ControlNodes".cm.axisCommand.cathodeMainPnP2AxisZ.posAbsolute[0] )
   END_RUNG
   RUNG wire#powerrail
      I_Contact( "Unit1.Em5.ControlNodes".gaugeRnR."step".action1[1640] )
      I_Contact( "Unit1.Em5.ControlNodes".gaugeRnR."step".action1[1940] )
      I_Contact( "Unit1.Em5.ControlNodes".gaugeRnR."step".action1[2040] )
      I_Contact( "Unit1.Em5.ControlNodes".gaugeRnR."step".action1[2240] )
      Not()
   END_RUNG wire#w1
   // the same network as SCL:
   #"cathodeMainPnP2AxisZ Position_"[0](Status := #unitStatus,   // "Position.LER_Axis"
                           commands := "Unit1.Em5.HmiInterface".cmCathodeMainPnP2AxisZ.commands,
                           interlockOk := "Unit1.Em5.ControlNodes".cm.Interlock.cathodeMainPnP2AxisZ.source.posAbsolute,
                           intOut := "Unit1.Em5.HmiInterface".intCondition.Axis_13.Position.intOut);
   #_w1 := (NOT (NOT "Unit1.Em5.ControlNodes".mainPnP."step".action1[1050] AND NOT "Unit1.Em5.ControlNodes".mainPnP."step".action1[125] AND NOT "Unit1.Em5.ControlNodes".mainPnP."step".action1[135] AND NOT "Unit1.Em5.ControlNodes".mainPnP."step".action1[145] AND NOT "Unit1.Em5.ControlNodes".mainPnP."step".action1[185] AND NOT "Unit1.Em5.ControlNodes".mainPnP."step".action1[210] AND NOT "Unit1.Em5.ControlNodes".mainPnP."step".action2[280] AND NOT "Unit1.Em5.ControlNodes".mainPnP."step".action1[310] AND NOT "Unit1.Em5.ControlNodes".mainPnP."step".action2[380]) OR NOT (NOT "Unit1.Em5.ControlNodes".gaugeRnR."step".action1[1640] AND NOT "Unit1.Em5.ControlNodes".gaugeRnR."step".action1[1940] AND NOT "Unit1.Em5.ControlNodes".gaugeRnR."step".action1[2040] AND NOT "Unit1.Em5.ControlNodes".gaugeRnR."step".action1[2240])) AND "Unit1.Em5.ControlNodes".cm.Interlock.cathodeMainPnP2AxisZ.source.posAbsolute[0];
   IF #_w1 THEN "Unit1.Em5.ControlNodes".cmCathodeMainPnP2AxisZ.commands.selectSetPosition := 0; END_IF;
   "Unit1.Em5.ControlNodes".cm.axisCommand.cathodeMainPnP2AxisZ.posAbsolute[0] := #_w1;
END_REGION

REGION Network 150: CmCathodeMainPnP2AxisZ Position Absolute Position1
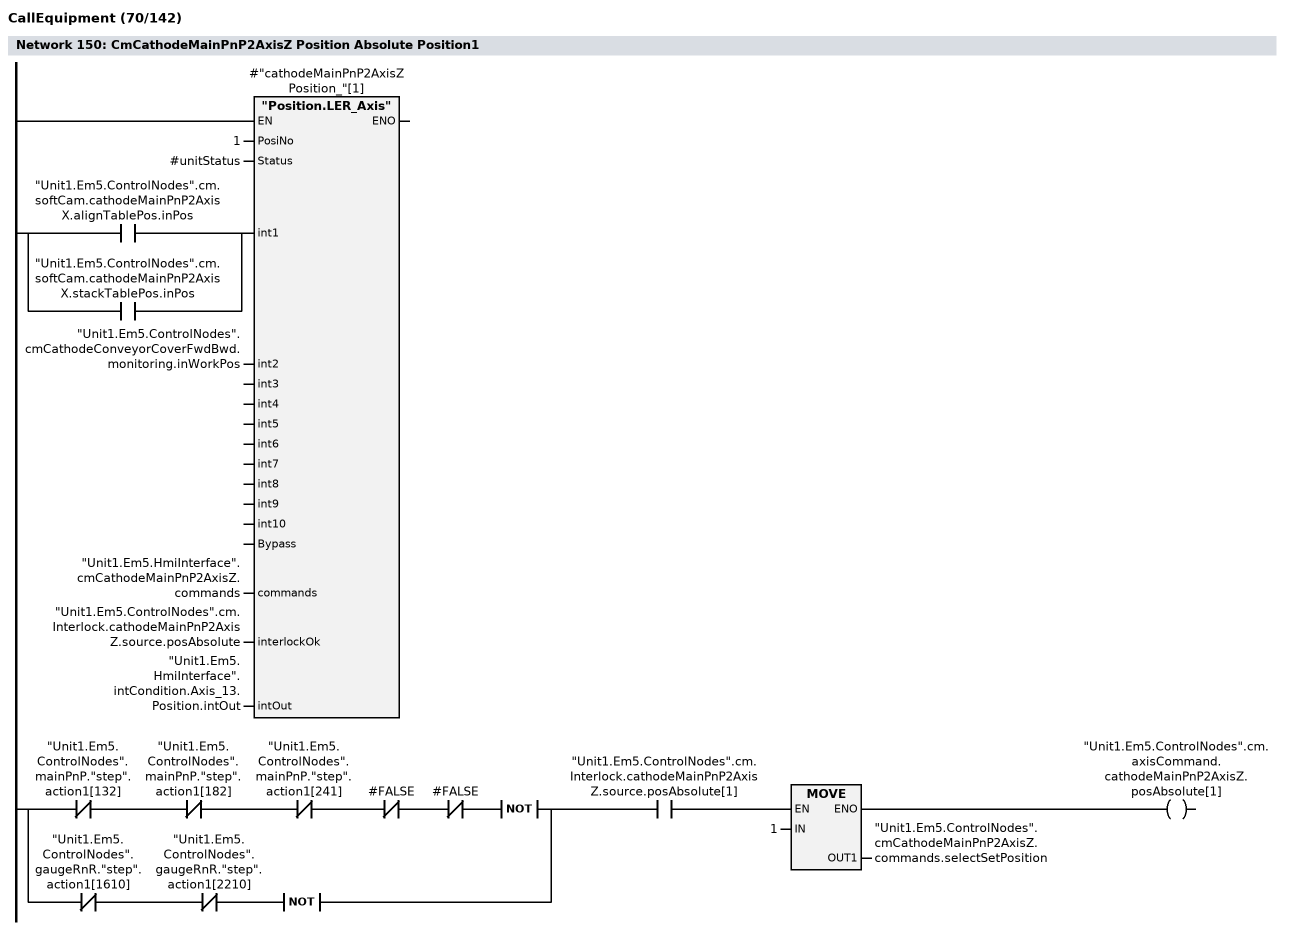
   RUNG wire#powerrail
      #"cathodeMainPnP2AxisZ Position_"[1](int1 := wire#w1, PosiNo := 1, Status := #unitStatus, int2 := "Unit1.Em5.ControlNodes".cmCathodeConveyorCoverFwdBwd.monitoring.inWorkPos, int3 :=, int4 :=, int5 :=, int6 :=, int7 :=, int8 :=, int9 :=, int10 :=, Bypass :=, commands := "Unit1.Em5.HmiInterface".cmCathodeMainPnP2AxisZ.commands, interlockOk := "Unit1.Em5.ControlNodes".cm.Interlock.cathodeMainPnP2AxisZ.source.posAbsolute, intOut := "Unit1.Em5.HmiInterface".intCondition.Axis_13.Position.intOut)
   END_RUNG
   RUNG wire#powerrail
      Contact( "Unit1.Em5.ControlNodes".cm.softCam.cathodeMainPnP2AxisX.alignTablePos.inPos )
   END_RUNG wire#w1
   RUNG wire#powerrail
      Contact( "Unit1.Em5.ControlNodes".cm.softCam.cathodeMainPnP2AxisX.stackTablePos.inPos )
   END_RUNG wire#w1
   RUNG wire#powerrail
      I_Contact( "Unit1.Em5.ControlNodes".mainPnP."step".action1[132] )
      I_Contact( "Unit1.Em5.ControlNodes".mainPnP."step".action1[182] )
      I_Contact( "Unit1.Em5.ControlNodes".mainPnP."step".action1[241] )
      I_Contact( #FALSE )
      I_Contact( #FALSE )
      Not()
      wire#w2
      Contact( "Unit1.Em5.ControlNodes".cm.Interlock.cathodeMainPnP2AxisZ.source.posAbsolute[1] )
      Move(in := 1, out1 => "Unit1.Em5.ControlNodes".cmCathodeMainPnP2AxisZ.commands.selectSetPosition)
      Coil( "Unit1.Em5.ControlNodes".cm.axisCommand.cathodeMainPnP2AxisZ.posAbsolute[1] )
   END_RUNG
   RUNG wire#powerrail
      I_Contact( "Unit1.Em5.ControlNodes".gaugeRnR."step".action1[1610] )
      I_Contact( "Unit1.Em5.ControlNodes".gaugeRnR."step".action1[2210] )
      Not()
   END_RUNG wire#w2
   // the same network as SCL:
   #"cathodeMainPnP2AxisZ Position_"[1](PosiNo := 1,   // "Position.LER_Axis"
                           Status := #unitStatus,
                           int1 := "Unit1.Em5.ControlNodes".cm.softCam.cathodeMainPnP2AxisX.alignTablePos.inPos OR "Unit1.Em5.ControlNodes".cm.softCam.cathodeMainPnP2AxisX.stackTablePos.inPos,
                           int2 := "Unit1.Em5.ControlNodes".cmCathodeConveyorCoverFwdBwd.monitoring.inWorkPos,
                           commands := "Unit1.Em5.HmiInterface".cmCathodeMainPnP2AxisZ.commands,
                           interlockOk := "Unit1.Em5.ControlNodes".cm.Interlock.cathodeMainPnP2AxisZ.source.posAbsolute,
                           intOut := "Unit1.Em5.HmiInterface".intCondition.Axis_13.Position.intOut);
   #_w1 := (NOT (NOT "Unit1.Em5.ControlNodes".mainPnP."step".action1[132] AND NOT "Unit1.Em5.ControlNodes".mainPnP."step".action1[182] AND NOT "Unit1.Em5.ControlNodes".mainPnP."step".action1[241] AND NOT #FALSE AND NOT #FALSE) OR NOT (NOT "Unit1.Em5.ControlNodes".gaugeRnR."step".action1[1610] AND NOT "Unit1.Em5.ControlNodes".gaugeRnR."step".action1[2210])) AND "Unit1.Em5.ControlNodes".cm.Interlock.cathodeMainPnP2AxisZ.source.posAbsolute[1];
   IF #_w1 THEN "Unit1.Em5.ControlNodes".cmCathodeMainPnP2AxisZ.commands.selectSetPosition := 1; END_IF;
   "Unit1.Em5.ControlNodes".cm.axisCommand.cathodeMainPnP2AxisZ.posAbsolute[1] := #_w1;
END_REGION

REGION Network 151: CmCathodeMainPnP2AxisZ Position Absolute Position2
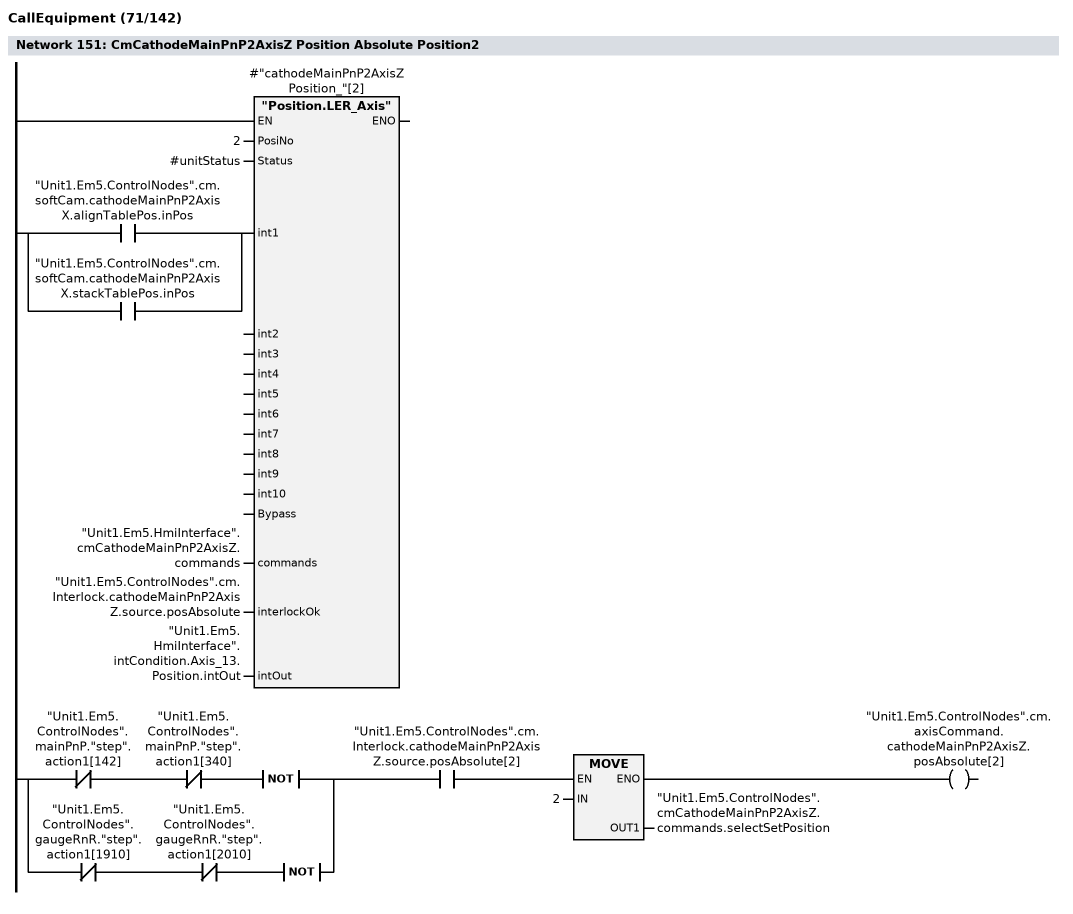
   RUNG wire#powerrail
      #"cathodeMainPnP2AxisZ Position_"[2](int1 := wire#w1, PosiNo := 2, Status := #unitStatus, int2 :=, int3 :=, int4 :=, int5 :=, int6 :=, int7 :=, int8 :=, int9 :=, int10 :=, Bypass :=, commands := "Unit1.Em5.HmiInterface".cmCathodeMainPnP2AxisZ.commands, interlockOk := "Unit1.Em5.ControlNodes".cm.Interlock.cathodeMainPnP2AxisZ.source.posAbsolute, intOut := "Unit1.Em5.HmiInterface".intCondition.Axis_13.Position.intOut)
   END_RUNG
   RUNG wire#powerrail
      Contact( "Unit1.Em5.ControlNodes".cm.softCam.cathodeMainPnP2AxisX.alignTablePos.inPos )
   END_RUNG wire#w1
   RUNG wire#powerrail
      Contact( "Unit1.Em5.ControlNodes".cm.softCam.cathodeMainPnP2AxisX.stackTablePos.inPos )
   END_RUNG wire#w1
   RUNG wire#powerrail
      I_Contact( "Unit1.Em5.ControlNodes".mainPnP."step".action1[142] )
      I_Contact( "Unit1.Em5.ControlNodes".mainPnP."step".action1[340] )
      Not()
      wire#w2
      Contact( "Unit1.Em5.ControlNodes".cm.Interlock.cathodeMainPnP2AxisZ.source.posAbsolute[2] )
      Move(in := 2, out1 => "Unit1.Em5.ControlNodes".cmCathodeMainPnP2AxisZ.commands.selectSetPosition)
      Coil( "Unit1.Em5.ControlNodes".cm.axisCommand.cathodeMainPnP2AxisZ.posAbsolute[2] )
   END_RUNG
   RUNG wire#powerrail
      I_Contact( "Unit1.Em5.ControlNodes".gaugeRnR."step".action1[1910] )
      I_Contact( "Unit1.Em5.ControlNodes".gaugeRnR."step".action1[2010] )
      Not()
   END_RUNG wire#w2
   // the same network as SCL:
   #"cathodeMainPnP2AxisZ Position_"[2](PosiNo := 2,   // "Position.LER_Axis"
                           Status := #unitStatus,
                           int1 := "Unit1.Em5.ControlNodes".cm.softCam.cathodeMainPnP2AxisX.alignTablePos.inPos OR "Unit1.Em5.ControlNodes".cm.softCam.cathodeMainPnP2AxisX.stackTablePos.inPos,
                           commands := "Unit1.Em5.HmiInterface".cmCathodeMainPnP2AxisZ.commands,
                           interlockOk := "Unit1.Em5.ControlNodes".cm.Interlock.cathodeMainPnP2AxisZ.source.posAbsolute,
                           intOut := "Unit1.Em5.HmiInterface".intCondition.Axis_13.Position.intOut);
   #_w1 := (NOT (NOT "Unit1.Em5.ControlNodes".mainPnP."step".action1[142] AND NOT "Unit1.Em5.ControlNodes".mainPnP."step".action1[340]) OR NOT (NOT "Unit1.Em5.ControlNodes".gaugeRnR."step".action1[1910] AND NOT "Unit1.Em5.ControlNodes".gaugeRnR."step".action1[2010])) AND "Unit1.Em5.ControlNodes".cm.Interlock.cathodeMainPnP2AxisZ.source.posAbsolute[2];
   IF #_w1 THEN "Unit1.Em5.ControlNodes".cmCathodeMainPnP2AxisZ.commands.selectSetPosition := 2; END_IF;
   "Unit1.Em5.ControlNodes".cm.axisCommand.cathodeMainPnP2AxisZ.posAbsolute[2] := #_w1;
END_REGION

REGION Network 152: CmCathodeMainPnP2AxisZ Position Absolute Position3
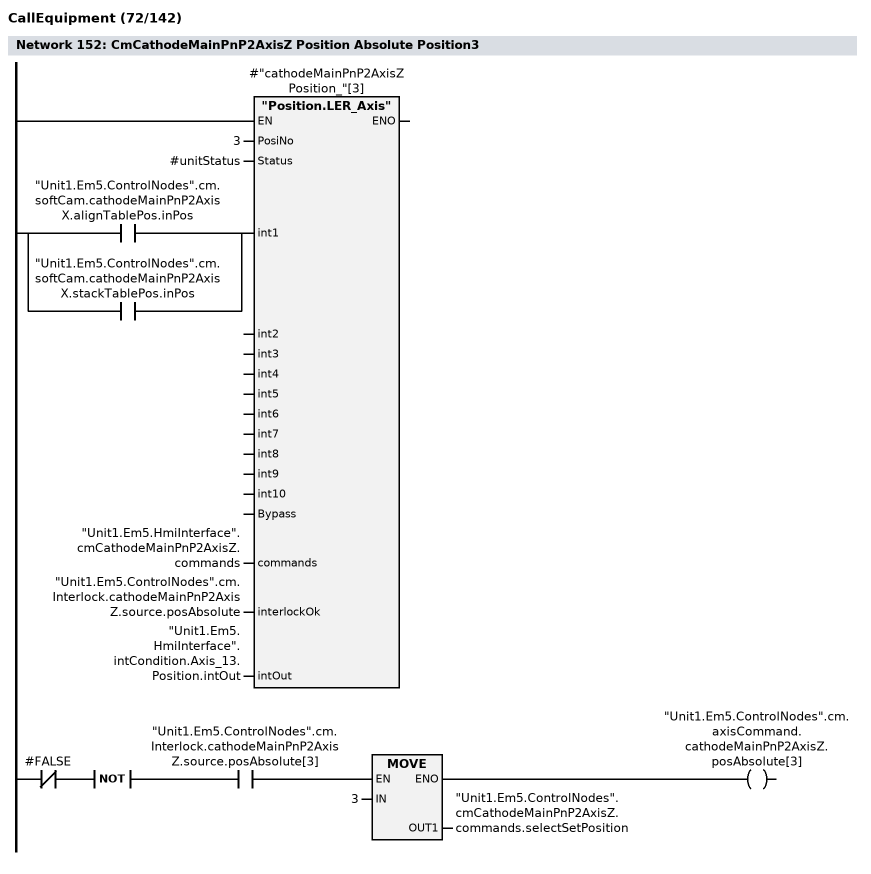
   RUNG wire#powerrail
      #"cathodeMainPnP2AxisZ Position_"[3](int1 := wire#w1, PosiNo := 3, Status := #unitStatus, int2 :=, int3 :=, int4 :=, int5 :=, int6 :=, int7 :=, int8 :=, int9 :=, int10 :=, Bypass :=, commands := "Unit1.Em5.HmiInterface".cmCathodeMainPnP2AxisZ.commands, interlockOk := "Unit1.Em5.ControlNodes".cm.Interlock.cathodeMainPnP2AxisZ.source.posAbsolute, intOut := "Unit1.Em5.HmiInterface".intCondition.Axis_13.Position.intOut)
   END_RUNG
   RUNG wire#powerrail
      Contact( "Unit1.Em5.ControlNodes".cm.softCam.cathodeMainPnP2AxisX.alignTablePos.inPos )
   END_RUNG wire#w1
   RUNG wire#powerrail
      Contact( "Unit1.Em5.ControlNodes".cm.softCam.cathodeMainPnP2AxisX.stackTablePos.inPos )
   END_RUNG wire#w1
   RUNG wire#powerrail
      I_Contact( #FALSE )
      Not()
      Contact( "Unit1.Em5.ControlNodes".cm.Interlock.cathodeMainPnP2AxisZ.source.posAbsolute[3] )
      Move(in := 3, out1 => "Unit1.Em5.ControlNodes".cmCathodeMainPnP2AxisZ.commands.selectSetPosition)
      Coil( "Unit1.Em5.ControlNodes".cm.axisCommand.cathodeMainPnP2AxisZ.posAbsolute[3] )
   END_RUNG
   // the same network as SCL:
   #"cathodeMainPnP2AxisZ Position_"[3](PosiNo := 3,   // "Position.LER_Axis"
                           Status := #unitStatus,
                           int1 := "Unit1.Em5.ControlNodes".cm.softCam.cathodeMainPnP2AxisX.alignTablePos.inPos OR "Unit1.Em5.ControlNodes".cm.softCam.cathodeMainPnP2AxisX.stackTablePos.inPos,
                           commands := "Unit1.Em5.HmiInterface".cmCathodeMainPnP2AxisZ.commands,
                           interlockOk := "Unit1.Em5.ControlNodes".cm.Interlock.cathodeMainPnP2AxisZ.source.posAbsolute,
                           intOut := "Unit1.Em5.HmiInterface".intCondition.Axis_13.Position.intOut);
   #_w1 := NOT (NOT #FALSE) AND "Unit1.Em5.ControlNodes".cm.Interlock.cathodeMainPnP2AxisZ.source.posAbsolute[3];
   IF #_w1 THEN "Unit1.Em5.ControlNodes".cmCathodeMainPnP2AxisZ.commands.selectSetPosition := 3; END_IF;
   "Unit1.Em5.ControlNodes".cm.axisCommand.cathodeMainPnP2AxisZ.posAbsolute[3] := #_w1;
END_REGION

REGION Network 153: CmCathodeMainPnP2AxisZ Position Absolute Position4
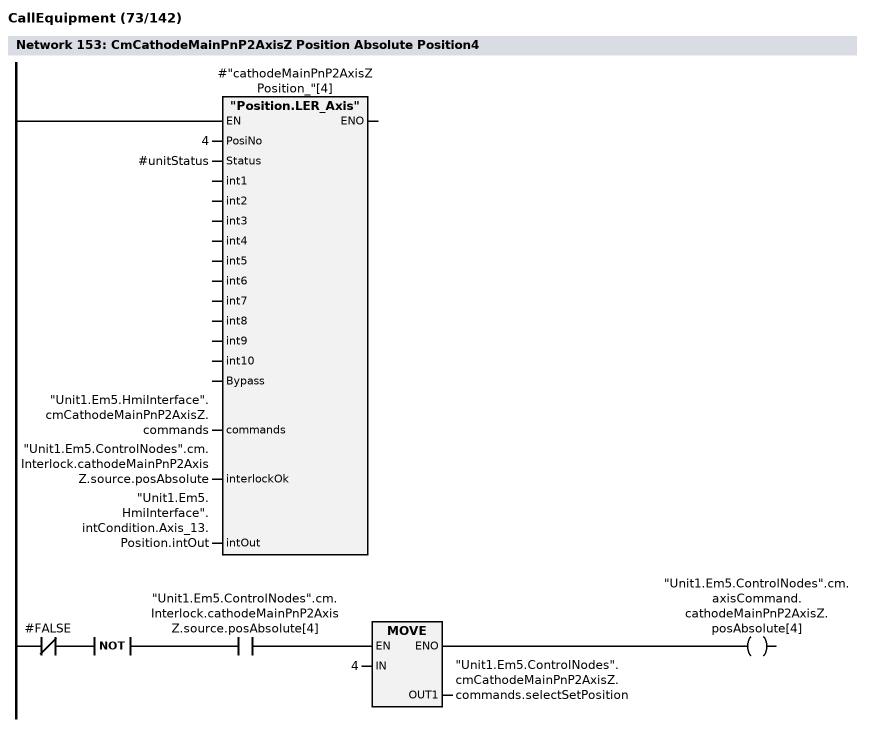
   RUNG wire#powerrail
      #"cathodeMainPnP2AxisZ Position_"[4](PosiNo := 4, Status := #unitStatus, int1 :=, int2 :=, int3 :=, int4 :=, int5 :=, int6 :=, int7 :=, int8 :=, int9 :=, int10 :=, Bypass :=, commands := "Unit1.Em5.HmiInterface".cmCathodeMainPnP2AxisZ.commands, interlockOk := "Unit1.Em5.ControlNodes".cm.Interlock.cathodeMainPnP2AxisZ.source.posAbsolute, intOut := "Unit1.Em5.HmiInterface".intCondition.Axis_13.Position.intOut)
   END_RUNG
   RUNG wire#powerrail
      I_Contact( #FALSE )
      Not()
      Contact( "Unit1.Em5.ControlNodes".cm.Interlock.cathodeMainPnP2AxisZ.source.posAbsolute[4] )
      Move(in := 4, out1 => "Unit1.Em5.ControlNodes".cmCathodeMainPnP2AxisZ.commands.selectSetPosition)
      Coil( "Unit1.Em5.ControlNodes".cm.axisCommand.cathodeMainPnP2AxisZ.posAbsolute[4] )
   END_RUNG
   // the same network as SCL:
   #"cathodeMainPnP2AxisZ Position_"[4](PosiNo := 4,   // "Position.LER_Axis"
                           Status := #unitStatus,
                           commands := "Unit1.Em5.HmiInterface".cmCathodeMainPnP2AxisZ.commands,
                           interlockOk := "Unit1.Em5.ControlNodes".cm.Interlock.cathodeMainPnP2AxisZ.source.posAbsolute,
                           intOut := "Unit1.Em5.HmiInterface".intCondition.Axis_13.Position.intOut);
   #_w1 := NOT (NOT #FALSE) AND "Unit1.Em5.ControlNodes".cm.Interlock.cathodeMainPnP2AxisZ.source.posAbsolute[4];
   IF #_w1 THEN "Unit1.Em5.ControlNodes".cmCathodeMainPnP2AxisZ.commands.selectSetPosition := 4; END_IF;
   "Unit1.Em5.ControlNodes".cm.axisCommand.cathodeMainPnP2AxisZ.posAbsolute[4] := #_w1;
END_REGION

REGION Network 154: CmCathodeMainPnP2AxisZ Position Absolute Position5
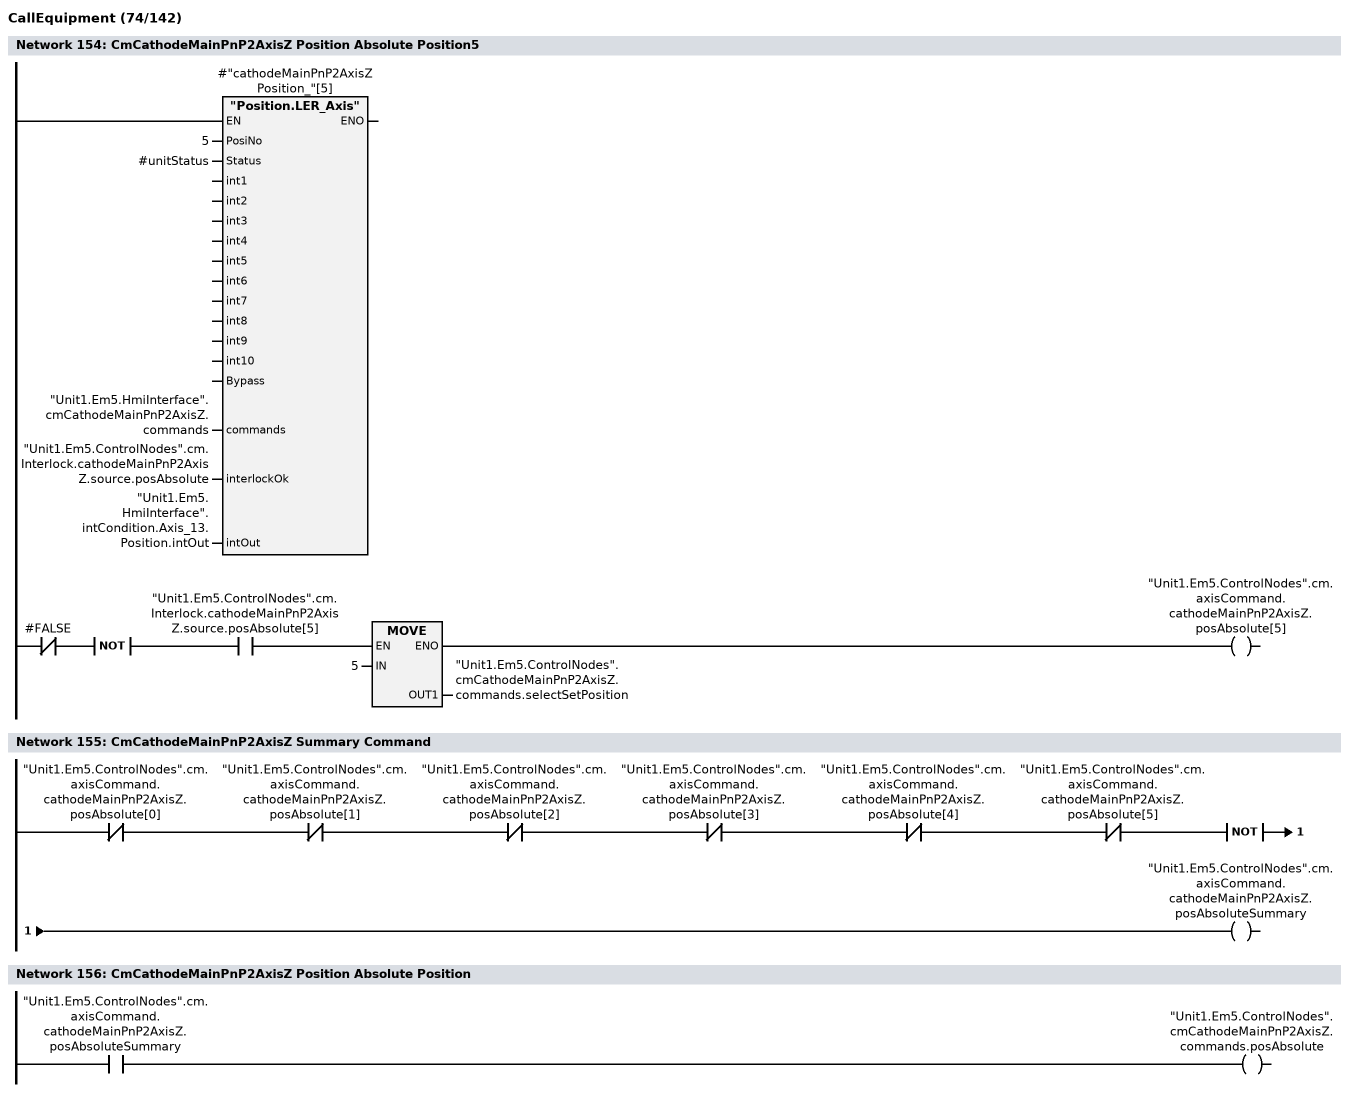
   RUNG wire#powerrail
      #"cathodeMainPnP2AxisZ Position_"[5](PosiNo := 5, Status := #unitStatus, int1 :=, int2 :=, int3 :=, int4 :=, int5 :=, int6 :=, int7 :=, int8 :=, int9 :=, int10 :=, Bypass :=, commands := "Unit1.Em5.HmiInterface".cmCathodeMainPnP2AxisZ.commands, interlockOk := "Unit1.Em5.ControlNodes".cm.Interlock.cathodeMainPnP2AxisZ.source.posAbsolute, intOut := "Unit1.Em5.HmiInterface".intCondition.Axis_13.Position.intOut)
   END_RUNG
   RUNG wire#powerrail
      I_Contact( #FALSE )
      Not()
      Contact( "Unit1.Em5.ControlNodes".cm.Interlock.cathodeMainPnP2AxisZ.source.posAbsolute[5] )
      Move(in := 5, out1 => "Unit1.Em5.ControlNodes".cmCathodeMainPnP2AxisZ.commands.selectSetPosition)
      Coil( "Unit1.Em5.ControlNodes".cm.axisCommand.cathodeMainPnP2AxisZ.posAbsolute[5] )
   END_RUNG
   // the same network as SCL:
   #"cathodeMainPnP2AxisZ Position_"[5](PosiNo := 5,   // "Position.LER_Axis"
                           Status := #unitStatus,
                           commands := "Unit1.Em5.HmiInterface".cmCathodeMainPnP2AxisZ.commands,
                           interlockOk := "Unit1.Em5.ControlNodes".cm.Interlock.cathodeMainPnP2AxisZ.source.posAbsolute,
                           intOut := "Unit1.Em5.HmiInterface".intCondition.Axis_13.Position.intOut);
   #_w1 := NOT (NOT #FALSE) AND "Unit1.Em5.ControlNodes".cm.Interlock.cathodeMainPnP2AxisZ.source.posAbsolute[5];
   IF #_w1 THEN "Unit1.Em5.ControlNodes".cmCathodeMainPnP2AxisZ.commands.selectSetPosition := 5; END_IF;
   "Unit1.Em5.ControlNodes".cm.axisCommand.cathodeMainPnP2AxisZ.posAbsolute[5] := #_w1;
END_REGION

REGION Network 155: CmCathodeMainPnP2AxisZ Summary Command
   RUNG wire#powerrail
      I_Contact( "Unit1.Em5.ControlNodes".cm.axisCommand.cathodeMainPnP2AxisZ.posAbsolute[0] )
      I_Contact( "Unit1.Em5.ControlNodes".cm.axisCommand.cathodeMainPnP2AxisZ.posAbsolute[1] )
      I_Contact( "Unit1.Em5.ControlNodes".cm.axisCommand.cathodeMainPnP2AxisZ.posAbsolute[2] )
      I_Contact( "Unit1.Em5.ControlNodes".cm.axisCommand.cathodeMainPnP2AxisZ.posAbsolute[3] )
      I_Contact( "Unit1.Em5.ControlNodes".cm.axisCommand.cathodeMainPnP2AxisZ.posAbsolute[4] )
      I_Contact( "Unit1.Em5.ControlNodes".cm.axisCommand.cathodeMainPnP2AxisZ.posAbsolute[5] )
      Not()
      Coil( "Unit1.Em5.ControlNodes".cm.axisCommand.cathodeMainPnP2AxisZ.posAbsoluteSummary )
   END_RUNG
   // the same network as SCL:
   "Unit1.Em5.ControlNodes".cm.axisCommand.cathodeMainPnP2AxisZ.posAbsoluteSummary := NOT (NOT "Unit1.Em5.ControlNodes".cm.axisCommand.cathodeMainPnP2AxisZ.posAbsolute[0] AND NOT "Unit1.Em5.ControlNodes".cm.axisCommand.cathodeMainPnP2AxisZ.posAbsolute[1] AND NOT "Unit1.Em5.ControlNodes".cm.axisCommand.cathodeMainPnP2AxisZ.posAbsolute[2] AND NOT "Unit1.Em5.ControlNodes".cm.axisCommand.cathodeMainPnP2AxisZ.posAbsolute[3] AND NOT "Unit1.Em5.ControlNodes".cm.axisCommand.cathodeMainPnP2AxisZ.posAbsolute[4] AND NOT "Unit1.Em5.ControlNodes".cm.axisCommand.cathodeMainPnP2AxisZ.posAbsolute[5]);
END_REGION

REGION Network 156: CmCathodeMainPnP2AxisZ Position Absolute Position
   RUNG wire#powerrail
      Contact( "Unit1.Em5.ControlNodes".cm.axisCommand.cathodeMainPnP2AxisZ.posAbsoluteSummary )
      Coil( "Unit1.Em5.ControlNodes".cmCathodeMainPnP2AxisZ.commands.posAbsolute )
   END_RUNG
   // the same network as SCL:
   "Unit1.Em5.ControlNodes".cmCathodeMainPnP2AxisZ.commands.posAbsolute := "Unit1.Em5.ControlNodes".cm.axisCommand.cathodeMainPnP2AxisZ.posAbsoluteSummary;
END_REGION

REGION Network 157: CmCathodeMainPnP1AxisZ Interlock Summary
